		IF arrCheckListForNestedSymbols[uiCounterCheckSubItemsInContentOfDoc] = arrContentOfDocument[uiCounterCkeckContenInSubItems_1].sSymbolName THEN
			IF arrContentOfDocument[uiCounterCkeckContenInSubItems_1].arrSubItemSymbolType[uiCounterCkeckContenInSubItems_2] <> 'BOOL' AND arrContentOfDocument[uiCounterCkeckContenInSubItems_1].arrSubItemSymbolType[uiCounterCkeckContenInSubItems_2] <> 'BYTE' AND
				arrContentOfDocument[uiCounterCkeckContenInSubItems_1].arrSubItemSymbolType[uiCounterCkeckContenInSubItems_2] <> 'WORD' AND arrContentOfDocument[uiCounterCkeckContenInSubItems_1].arrSubItemSymbolType[uiCounterCkeckContenInSubItems_2] <> 'DWORD' AND
					arrContentOfDocument[uiCounterCkeckContenInSubItems_1].arrSubItemSymbolType[uiCounterCkeckContenInSubItems_2] <> 'SINT' AND arrContentOfDocument[uiCounterCkeckContenInSubItems_1].arrSubItemSymbolType[uiCounterCkeckContenInSubItems_2] <> 'USINT' AND
						arrContentOfDocument[uiCounterCkeckContenInSubItems_1].arrSubItemSymbolType[uiCounterCkeckContenInSubItems_2] <> 'INT' AND arrContentOfDocument[uiCounterCkeckContenInSubItems_1].arrSubItemSymbolType[uiCounterCkeckContenInSubItems_2] <> 'UINT' AND
							arrContentOfDocument[uiCounterCkeckContenInSubItems_1].arrSubItemSymbolType[uiCounterCkeckContenInSubItems_2] <> 'DINT' AND arrContentOfDocument[uiCounterCkeckContenInSubItems_1].arrSubItemSymbolType[uiCounterCkeckContenInSubItems_2] <> 'UDINT' AND
								arrContentOfDocument[uiCounterCkeckContenInSubItems_1].arrSubItemSymbolType[uiCounterCkeckContenInSubItems_2] <> 'LINT' AND arrContentOfDocument[uiCounterCkeckContenInSubItems_1].arrSubItemSymbolType[uiCounterCkeckContenInSubItems_2] <> 'ULINT' AND
									arrContentOfDocument[uiCounterCkeckContenInSubItems_1].arrSubItemSymbolType[uiCounterCkeckContenInSubItems_2] <> 'LWORD' AND arrContentOfDocument[uiCounterCkeckContenInSubItems_1].arrSubItemSymbolType[uiCounterCkeckContenInSubItems_2] <> 'REAL' AND
										arrContentOfDocument[uiCounterCkeckContenInSubItems_1].arrSubItemSymbolType[uiCounterCkeckContenInSubItems_2] <> 'LREAL' AND arrContentOfDocument[uiCounterCkeckContenInSubItems_1].arrSubItemSymbolType[uiCounterCkeckContenInSubItems_2] <> 'STRING(30)' AND
											arrContentOfDocument[uiCounterCkeckContenInSubItems_1].arrSubItemSymbolType[uiCounterCkeckContenInSubItems_2] <> 'TIME' AND arrContentOfDocument[uiCounterCkeckContenInSubItems_1].arrSubItemSymbolType[uiCounterCkeckContenInSubItems_2] <> 'TIME_OF_DAY' AND
												arrContentOfDocument[uiCounterCkeckContenInSubItems_1].arrSubItemSymbolType[uiCounterCkeckContenInSubItems_2] <> 'DATE' AND arrContentOfDocument[uiCounterCkeckContenInSubItems_1].arrSubItemSymbolType[uiCounterCkeckContenInSubItems_2] <> 'DATE_AND_TIME' AND 
			FIND(arrContentOfDocument[uiCounterCkeckContenInSubItems_1].arrSubItemSymbolType[uiCounterCkeckContenInSubItems_2],'OF BOOL') = 0 AND FIND(arrContentOfDocument[uiCounterCkeckContenInSubItems_1].arrSubItemSymbolType[uiCounterCkeckContenInSubItems_2],'OF BYTE') = 0 AND
				FIND(arrContentOfDocument[uiCounterCkeckContenInSubItems_1].arrSubItemSymbolType[uiCounterCkeckContenInSubItems_2],'OF WORD') = 0 AND FIND(arrContentOfDocument[uiCounterCkeckContenInSubItems_1].arrSubItemSymbolType[uiCounterCkeckContenInSubItems_2],'OF DWORD') = 0 AND
					FIND(arrContentOfDocument[uiCounterCkeckContenInSubItems_1].arrSubItemSymbolType[uiCounterCkeckContenInSubItems_2],'OF SINT') = 0 AND FIND(arrContentOfDocument[uiCounterCkeckContenInSubItems_1].arrSubItemSymbolType[uiCounterCkeckContenInSubItems_2],'OF USINT') = 0 AND 
						FIND(arrContentOfDocument[uiCounterCkeckContenInSubItems_1].arrSubItemSymbolType[uiCounterCkeckContenInSubItems_2],'OF INT') = 0 AND FIND(arrContentOfDocument[uiCounterCkeckContenInSubItems_1].arrSubItemSymbolType[uiCounterCkeckContenInSubItems_2],'OF UINT') = 0 AND
							FIND(arrContentOfDocument[uiCounterCkeckContenInSubItems_1].arrSubItemSymbolType[uiCounterCkeckContenInSubItems_2],'OF DINT') = 0 AND FIND(arrContentOfDocument[uiCounterCkeckContenInSubItems_1].arrSubItemSymbolType[uiCounterCkeckContenInSubItems_2],'OF UDINT') = 0 AND
								FIND(arrContentOfDocument[uiCounterCkeckContenInSubItems_1].arrSubItemSymbolType[uiCounterCkeckContenInSubItems_2],'OF LINT') = 0 AND FIND(arrContentOfDocument[uiCounterCkeckContenInSubItems_1].arrSubItemSymbolType[uiCounterCkeckContenInSubItems_2],'OF ULINT') = 0 AND
									FIND(arrContentOfDocument[uiCounterCkeckContenInSubItems_1].arrSubItemSymbolType[uiCounterCkeckContenInSubItems_2],'OF LWORD') = 0 AND FIND(arrContentOfDocument[uiCounterCkeckContenInSubItems_1].arrSubItemSymbolType[uiCounterCkeckContenInSubItems_2],'OF REAL') = 0 AND
										FIND(arrContentOfDocument[uiCounterCkeckContenInSubItems_1].arrSubItemSymbolType[uiCounterCkeckContenInSubItems_2],'OF LREAL') = 0 AND FIND(arrContentOfDocument[uiCounterCkeckContenInSubItems_1].arrSubItemSymbolType[uiCounterCkeckContenInSubItems_2],'OF STRING(30)') = 0 AND
											FIND(arrContentOfDocument[uiCounterCkeckContenInSubItems_1].arrSubItemSymbolType[uiCounterCkeckContenInSubItems_2],'OF TIME') = 0 AND FIND(arrContentOfDocument[uiCounterCkeckContenInSubItems_1].arrSubItemSymbolType[uiCounterCkeckContenInSubItems_2],'OF TIME_OF_DAY') = 0 AND
												FIND(arrContentOfDocument[uiCounterCkeckContenInSubItems_1].arrSubItemSymbolType[uiCounterCkeckContenInSubItems_2],'OF DATE') = 0 AND FIND(arrContentOfDocument[uiCounterCkeckContenInSubItems_1].arrSubItemSymbolType[uiCounterCkeckContenInSubItems_2],'OF DATE_AND_TIME') = 0 AND
			arrContentOfDocument[uiCounterCkeckContenInSubItems_1].arrSubItemSymbolType[uiCounterCkeckContenInSubItems_2] <> '' THEN 
				iStateParseDocument := 200;
					udiErrorCode := 117;
			END_IF	
		END_IF
		
		IF uiCounterCheckSubItemsInContentOfDoc >= uiCounterListForFBorStruct AND uiCounterCkeckContenInSubItems_1 >= uiCounterInProgressFromDocument AND uiCounterCkeckContenInSubItems_2 >= Constants_Communicator.uiArraySizeOfMarkedSubItems AND iStateParseDocument = 105 THEN 
			iStateParseDocument := 106; byProgress := byProgress + 1;
				uiCounterCheckSubItemsInContentOfDoc := 0; uiCounterCkeckContenInSubItems_1 := 0; uiCounterCkeckContenInSubItems_2 := 0;
		END_IF
		
	106://Check in Sub Items for no standart Datatypes in Array	
		uiCounterCkeckContenInSubItems_2 := uiCounterCkeckContenInSubItems_2 + 1;
		
		IF uiCounterCkeckContenInSubItems_2 > Constants_Communicator.uiArraySizeOfMarkedSubItems THEN uiCounterCkeckContenInSubItems_1 := uiCounterCkeckContenInSubItems_1 + 1; END_IF
			
		IF uiCounterCkeckContenInSubItems_2 > Constants_Communicator.uiArraySizeOfMarkedSubItems AND uiCounterCkeckContenInSubItems_1 > uiCounterInProgressFromDocument THEN uiCounterCheckSubItemsInContentOfDoc := uiCounterCheckSubItemsInContentOfDoc + 1; END_IF	

		IF uiCounterCkeckContenInSubItems_1 > uiCounterInProgressFromDocument THEN uiCounterCkeckContenInSubItems_1 := 1; END_IF	
		IF uiCounterCkeckContenInSubItems_2 > Constants_Communicator.uiArraySizeOfMarkedSubItems THEN uiCounterCkeckContenInSubItems_2 := 1; END_IF
	
		uiCounterCkeckContenInSubItems_2 := LIMIT(1,uiCounterCkeckContenInSubItems_2,Constants_Communicator.uiArraySizeOfMarkedSubItems);	
		uiCounterCheckSubItemsInContentOfDoc := LIMIT(1,uiCounterCheckSubItemsInContentOfDoc,Constants_Communicator.uiArraySizeOfSubItems);
		uiCounterCkeckContenInSubItems_1 := LIMIT(1,uiCounterCkeckContenInSubItems_1,Constants_Communicator.uiArraySizeOfSubItems);
		
		//Array with no Standart Datatype
		IF FIND(arrContentOfDocument[uiCounterCkeckContenInSubItems_1].arrSubItemSymbolType[uiCounterCkeckContenInSubItems_2],'ARRAY') = 1 AND 
			FIND(arrContentOfDocument[uiCounterCkeckContenInSubItems_1].arrSubItemSymbolType[uiCounterCkeckContenInSubItems_2],'OF BOOL') = 0 AND FIND(arrContentOfDocument[uiCounterCkeckContenInSubItems_1].arrSubItemSymbolType[uiCounterCkeckContenInSubItems_2],'OF BYTE') = 0 AND
				FIND(arrContentOfDocument[uiCounterCkeckContenInSubItems_1].arrSubItemSymbolType[uiCounterCkeckContenInSubItems_2],'OF WORD') = 0 AND FIND(arrContentOfDocument[uiCounterCkeckContenInSubItems_1].arrSubItemSymbolType[uiCounterCkeckContenInSubItems_2],'OF DWORD') = 0 AND
					FIND(arrContentOfDocument[uiCounterCkeckContenInSubItems_1].arrSubItemSymbolType[uiCounterCkeckContenInSubItems_2],'OF SINT') = 0 AND FIND(arrContentOfDocument[uiCounterCkeckContenInSubItems_1].arrSubItemSymbolType[uiCounterCkeckContenInSubItems_2],'OF USINT') = 0 AND 
						FIND(arrContentOfDocument[uiCounterCkeckContenInSubItems_1].arrSubItemSymbolType[uiCounterCkeckContenInSubItems_2],'OF INT') = 0 AND FIND(arrContentOfDocument[uiCounterCkeckContenInSubItems_1].arrSubItemSymbolType[uiCounterCkeckContenInSubItems_2],'OF UINT') = 0 AND
							FIND(arrContentOfDocument[uiCounterCkeckContenInSubItems_1].arrSubItemSymbolType[uiCounterCkeckContenInSubItems_2],'OF DINT') = 0 AND FIND(arrContentOfDocument[uiCounterCkeckContenInSubItems_1].arrSubItemSymbolType[uiCounterCkeckContenInSubItems_2],'OF UDINT') = 0 AND
								FIND(arrContentOfDocument[uiCounterCkeckContenInSubItems_1].arrSubItemSymbolType[uiCounterCkeckContenInSubItems_2],'OF LINT') = 0 AND FIND(arrContentOfDocument[uiCounterCkeckContenInSubItems_1].arrSubItemSymbolType[uiCounterCkeckContenInSubItems_2],'OF ULINT') = 0 AND
									FIND(arrContentOfDocument[uiCounterCkeckContenInSubItems_1].arrSubItemSymbolType[uiCounterCkeckContenInSubItems_2],'OF LWORD') = 0 AND FIND(arrContentOfDocument[uiCounterCkeckContenInSubItems_1].arrSubItemSymbolType[uiCounterCkeckContenInSubItems_2],'OF REAL') = 0 AND
										FIND(arrContentOfDocument[uiCounterCkeckContenInSubItems_1].arrSubItemSymbolType[uiCounterCkeckContenInSubItems_2],'OF LREAL') = 0 AND FIND(arrContentOfDocument[uiCounterCkeckContenInSubItems_1].arrSubItemSymbolType[uiCounterCkeckContenInSubItems_2],'OF STRING(30)') = 0 AND
											FIND(arrContentOfDocument[uiCounterCkeckContenInSubItems_1].arrSubItemSymbolType[uiCounterCkeckContenInSubItems_2],'OF TIME') = 0 AND FIND(arrContentOfDocument[uiCounterCkeckContenInSubItems_1].arrSubItemSymbolType[uiCounterCkeckContenInSubItems_2],'OF TIME_OF_DAY') = 0 AND
												FIND(arrContentOfDocument[uiCounterCkeckContenInSubItems_1].arrSubItemSymbolType[uiCounterCkeckContenInSubItems_2],'OF DATE') = 0 AND FIND(arrContentOfDocument[uiCounterCkeckContenInSubItems_1].arrSubItemSymbolType[uiCounterCkeckContenInSubItems_2],'OF DATE_AND_TIME') = 0 AND
			arrContentOfDocument[uiCounterCkeckContenInSubItems_1].arrSubItemSymbolType[uiCounterCkeckContenInSubItems_2] <> '' THEN 
				iStateParseDocument := 200;
					udiErrorCode := 118;
		END_IF
	
		IF uiCounterCheckSubItemsInContentOfDoc >= uiCounterListForFBorStruct AND uiCounterCkeckContenInSubItems_1 >= uiCounterInProgressFromDocument AND uiCounterCkeckContenInSubItems_2 >= Constants_Communicator.uiArraySizeOfMarkedSubItems AND iStateParseDocument = 106 THEN 
			iStateParseDocument := 0; byProgress := 100; bDone := TRUE; uiFoundItems := uiCounterInProgressFromDocument; 
		END_IF
		
	200://Error
		IF udiErrorCode = 101 OR udiErrorCode = 102 OR udiErrorCode = 103 OR udiErrorCode = 108 OR udiErrorCode = 109 OR udiErrorCode = 110 OR udiErrorCode = 3 OR udiErrorCode = 4 THEN sSymbolNameWithError := sSymbolName; END_IF
			IF udiErrorCode = 104 THEN sSymbolNameWithError := CONCAT(CONCAT(sSymbolName,'.'),sNameSubItem); END_IF 
				IF ((udiErrorCode = 111 OR udiErrorCode = 112) AND uiCounterWantedSymbolInProgress <= 1 AND uiSubItemArrayInProgress <= 2) THEN 
					sSymbolNameWithError := CONCAT(CONCAT(arrContentOfDocument[1].sSymbolName,'.'),arrContentOfDocument[1].arrSubItemName[1]); 
				END_IF
					IF ((udiErrorCode = 111 OR udiErrorCode = 112) AND uiCounterWantedSymbolInProgress > 1 AND uiSubItemArrayInProgress <= 2) THEN 
						sSymbolNameWithError := CONCAT(CONCAT(arrContentOfDocument[uiCounterWantedSymbolInProgress].sSymbolName,'.'),arrContentOfDocument[uiCounterWantedSymbolInProgress].arrSubItemName[1]); 
					END_IF
						IF ((udiErrorCode = 111 OR udiErrorCode = 112) AND uiCounterWantedSymbolInProgress <= 1 AND uiSubItemArrayInProgress > 2) THEN 
							sSymbolNameWithError := CONCAT(CONCAT(arrContentOfDocument[1].sSymbolName,'.'),arrContentOfDocument[1].arrSubItemName[uiSubItemArrayInProgress - 1]); 
						END_IF
							IF ((udiErrorCode = 111 OR udiErrorCode = 112) AND uiCounterWantedSymbolInProgress > 1 AND uiSubItemArrayInProgress > 2) THEN 
								sSymbolNameWithError := CONCAT(CONCAT(arrContentOfDocument[uiCounterWantedSymbolInProgress].sSymbolName,'.'),arrContentOfDocument[uiCounterWantedSymbolInProgress].arrSubItemName[uiSubItemArrayInProgress - 1]); 
							END_IF
								IF udiErrorCode = 115 OR udiErrorCode = 116 OR udiErrorCode = 117 THEN sSymbolNameWithError := arrCheckListForNestedSymbols[uiCounterCheckSubItemsInContentOfDoc]; END_IF 
									IF udiErrorCode = 118 THEN sSymbolNameWithError := arrContentOfDocument[uiCounterCkeckContenInSubItems_1].sSymbolName; END_IF 
		bError := TRUE;
			iStateParseDocument := 0;
			
END_CASE

//Save position
IF eSavePositionTMCFile = eSavePositionFile.ePostionC THEN fbFileOpen.sPathName := CONCAT(CONCAT('C:\TwinCAT\3.1\Config\TMC\',TwinCAT_SystemInfoVarList._AppInfo.ProjectName),'.tmc'); END_IF
IF eSavePositionTMCFile = eSavePositionFile.ePostionHardDisk THEN fbFileOpen.sPathName := CONCAT(CONCAT('Hard Disk\TwinCAT\3.1\Config\TMC\',TwinCAT_SystemInfoVarList._AppInfo.ProjectName),'.tmc'); END_IF

fbFileOpen(
	sNetId:= , 
	sPathName:= , 
	nMode:= FOPEN_MODEREAD OR FOPEN_MODETEXT, 
	ePath:= PATH_GENERIC, 
	bExecute:= , 
	tTimeout:= T#5S, 
	bBusy=> , 
	bError=> , 
	nErrId=> , 
	hFile=> );

FPErrorOpen(CLK:= fbFileOpen.bError, Q=> );
	
fbFileGet(
	sNetId:= , 
	hFile:= fbFileOpen.hFile, 
	bExecute:= , 
	tTimeout:= T#5S, 
	bBusy=> , 
	bError=> , 
	nErrId=> , 
	sLine=> , 
	bEOF=> );

FPErrorGet(CLK:= fbFileGet.bError, Q=> );

fbFileTell(
	sNetId:= , 
	hFile:= fbFileOpen.hFile, 
	bExecute:= , 
	tTimeout:= T#5S, 
	bBusy=> , 
	bError=> , 
	nErrId=> , 
	nSeekPos=> );

FPErrorTell(CLK:= fbFileTell.bError, Q=> );	

fbFileSeek(
	sNetId:= , 
	hFile:= fbFileOpen.hFile, 
	nSeekPos:= , 
	eOrigin:= SEEK_END, 
	bExecute:= , 
	tTimeout:= T#5S, 
	bBusy=> , 
	bError=> , 
	nErrId=> );

FPErrorSeek(CLK:= fbFileSeek.bError, Q=> );
	
fbFileClose(
	sNetId:= , 
	hFile:= fbFileOpen.hFile, 
	bExecute:= , 
	tTimeout:= T#5S, 
	bBusy=> , 
	bError=> , 
	nErrId=> );
	
FPErrorClose(CLK:= fbFileClose.bError, Q=> );	

//Progress
IF iStateParseDocument > 3 AND iStateParseDocument < 100 AND diEndPositionInDocument > 0 THEN
	byProgress := REAL_TO_BYTE(F_Scalvalue(x:= DINT_TO_REAL(fbFileTell.nSeekPos), x1:= 0, y1:= 0, x2:= DINT_TO_REAL(diEndPositionInDocument), y2:= 100));
		IF byProgress >= 5 THEN
			byProgress := byProgress - 5;
		ELSE
			byProgress := 0;
		END_IF
END_IF

END_FUNCTION_BLOCK

// ---- General/FUNs Internal/F_Scalvalue.TcPOU
{attribute 'conditionalshow'}
FUNCTION F_Scalvalue : REAL
VAR_INPUT
	{attribute 'hide'}
	x 	: REAL;		//Scale Value
	{attribute 'hide'}
	x1	: REAL;		//Point 1, x-coordinate
	{attribute 'hide'}
	y1	: REAL;		//Point 1, y-coordinate
	{attribute 'hide'}
	x2	: REAL;		//Point 2, x-coordinate
	{attribute 'hide'}
	y2	: REAL;		//Point 2, y-coordinate
END_VAR
VAR
	{attribute 'hide'}
	k, d: REAL;		//Calculation points
END_VAR

//Slope of the straight line
IF x2 <> x1 THEN
	k:=	(y2 - y1) / (x2 - x1);
ELSE
	//Avoid division by 0
	k:= 1;
END_IF
//Intersection with the Y axis
d:= y1 - (k * x1);

//Output scaling
F_Scalvalue:= (k * x) + d;

END_FUNCTION

// ---- Communicator/FBs Internal/FB_VarInfo_ErrorCodes.TcPOU
{attribute 'conditionalshow'}
FUNCTION_BLOCK FB_VarInfo_ErrorCodes
VAR_INPUT
	{attribute 'hide'}
	bErrorADS				: BOOL;											//Error ADS function
	{attribute 'hide'}
	bErrorIntern			: BOOL;											//Other Error
	{attribute 'hide'}
	udiErrorCodeADS			: UDINT;										//Error Code ADS function
	{attribute 'hide'}
	udiErrorCodesIntern		: UDINT;										//Error code from other errors
END_VAR
VAR_OUTPUT
	{attribute 'hide'}
	udiErrorCodeADS_Out		: UDINT;										//ADS return code
	{attribute 'hide'}
	bError					: BOOL;											//Error flag
	eErrorVarInfo_Out		: eErrorVarInfo;								//Enum with Error from the Var Info function
END_VAR
VAR
END_VAR

//Creator : Kai Ebensperger
//Company : Lynus AG
//Date : 01.04.2020
//Version : 1.0.0.0

//With this function its possible to give out a Error return code from the ads or the internal codes from the read variable info function
//Directly from the ads
IF bErrorIntern OR bErrorADS THEN bError := TRUE; ELSE bError := FALSE; END_IF
	IF bErrorADS THEN udiErrorCodeADS_Out := udiErrorCodeADS; ELSE udiErrorCodeADS_Out := 0; END_IF

//Internal error codes from Var Info
IF bErrorIntern AND udiErrorCodesIntern = 1 THEN eErrorVarInfo_Out := eErrorVarInfo.eArraySizeError; 
ELSIF bErrorIntern AND udiErrorCodesIntern = 2 THEN eErrorVarInfo_Out := eErrorVarInfo.eTimoutError;
ELSIF bErrorIntern AND udiErrorCodesIntern = 3 THEN eErrorVarInfo_Out := eErrorVarInfo.eCommentLenghtError;
ELSIF bErrorIntern AND udiErrorCodesIntern = 4 THEN eErrorVarInfo_Out := eErrorVarInfo.eCommentDescriptionError;
ELSIF bErrorIntern AND udiErrorCodesIntern = 5 THEN eErrorVarInfo_Out := eErrorVarInfo.eSymbolTypeError;
ELSIF bErrorIntern AND udiErrorCodesIntern = 6 THEN eErrorVarInfo_Out := eErrorVarInfo.eSymbolNameToLongError; 
ELSIF bErrorIntern AND udiErrorCodesIntern = 7 THEN eErrorVarInfo_Out := eErrorVarInfo.eReadWriteFunctionToMuch; 
ELSIF bErrorIntern AND udiErrorCodesIntern = 8 THEN eErrorVarInfo_Out := eErrorVarInfo.eVarInfoFunctionToMuch;
ELSIF bErrorIntern AND udiErrorCodesIntern = 9 THEN eErrorVarInfo_Out := eErrorVarInfo.eSendReceiveFunctionToMuch; 
ELSIF bErrorIntern AND udiErrorCodesIntern = 10 THEN eErrorVarInfo_Out := eErrorVarInfo.eMoreReadWriteFuctionsAsSymbols;
ELSIF bErrorIntern AND udiErrorCodesIntern = 11 THEN eErrorVarInfo_Out := eErrorVarInfo.eNoTMCFileSelected;
ELSIF bErrorIntern AND udiErrorCodesIntern = 12 THEN eErrorVarInfo_Out := eErrorVarInfo.eArrayWithNoStandartDatatype; 
ELSIF bErrorIntern AND udiErrorCodesIntern = 13 THEN eErrorVarInfo_Out := eErrorVarInfo.eSymbolNotFoundInTMCFile; 
ELSIF bErrorIntern AND udiErrorCodesIntern = 14 THEN eErrorVarInfo_Out := eErrorVarInfo.eSymbolNameWithSubItemIsToLong;	
ELSIF bErrorIntern AND udiErrorCodesIntern = 15 THEN eErrorVarInfo_Out := eErrorVarInfo.eToMuchSubItemsInSymbol;
ELSIF bErrorIntern AND udiErrorCodesIntern = 16 THEN eErrorVarInfo_Out := eErrorVarInfo.eToMuchSymbols;
ELSIF bErrorIntern AND udiErrorCodesIntern = 17 THEN eErrorVarInfo_Out := eErrorVarInfo.eSubItemsInfoError;
ELSIF bErrorIntern AND udiErrorCodesIntern = 18 THEN eErrorVarInfo_Out := eErrorVarInfo.eNoSendReceiveFunction;
ELSIF bErrorIntern AND udiErrorCodesIntern = 19 THEN eErrorVarInfo_Out := eErrorVarInfo.eNoReadWriteFunction;
ELSIF bErrorIntern AND udiErrorCodesIntern = 20 THEN eErrorVarInfo_Out := eErrorVarInfo.eNoSymbolsFound;	
//Internal error codes from Parse Function	
ELSIF bErrorIntern AND udiErrorCodesIntern = 100 THEN eErrorVarInfo_Out := eErrorVarInfo.eTMCFileTimoutError;
ELSIF bErrorIntern AND udiErrorCodesIntern = 101 THEN eErrorVarInfo_Out := eErrorVarInfo.eTMCFileContentOfSymbolIsToBig;
ELSIF bErrorIntern AND udiErrorCodesIntern = 102 THEN eErrorVarInfo_Out := eErrorVarInfo.eTMCFileSymbolNameToLongError;	
ELSIF bErrorIntern AND udiErrorCodesIntern = 103 THEN eErrorVarInfo_Out := eErrorVarInfo.eTMCFileToMuchSubItemsInOneSymbol;
ELSIF bErrorIntern AND udiErrorCodesIntern = 104 THEN eErrorVarInfo_Out := eErrorVarInfo.eTMCFileSubItemNameToLongError;
ELSIF bErrorIntern AND udiErrorCodesIntern = 105 THEN eErrorVarInfo_Out := eErrorVarInfo.eTMCFileErrorWhenOpeningTheFile;
ELSIF bErrorIntern AND udiErrorCodesIntern = 106 THEN eErrorVarInfo_Out := eErrorVarInfo.eTMCFileErrorWhenReadingTheFile;
ELSIF bErrorIntern AND udiErrorCodesIntern = 107 THEN eErrorVarInfo_Out := eErrorVarInfo.eTMCFileErrorWhenClosingTheFile;
ELSIF bErrorIntern AND udiErrorCodesIntern = 108 THEN eErrorVarInfo_Out := eErrorVarInfo.eTMCFileToMuchNoStandartDatatypes;	
ELSIF bErrorIntern AND udiErrorCodesIntern = 109 THEN eErrorVarInfo_Out := eErrorVarInfo.eTMCFileEnumNameToLongError;
ELSIF bErrorIntern AND udiErrorCodesIntern = 110 THEN eErrorVarInfo_Out := eErrorVarInfo.eTMCFileEnumIndexToMuchSizes;
ELSIF bErrorIntern AND udiErrorCodesIntern = 111 THEN eErrorVarInfo_Out := eErrorVarInfo.eTMCFileArraySizeError;
ELSIF bErrorIntern AND udiErrorCodesIntern = 112 THEN eErrorVarInfo_Out := eErrorVarInfo.eTMCFileStringSizeError;
ELSIF bErrorIntern AND udiErrorCodesIntern = 113 THEN eErrorVarInfo_Out := eErrorVarInfo.eTMCFileCheckPositionError;
ELSIF bErrorIntern AND udiErrorCodesIntern = 114 THEN eErrorVarInfo_Out := eErrorVarInfo.eTMCFileSearchPositionError;
ELSIF bErrorIntern AND udiErrorCodesIntern = 115 THEN eErrorVarInfo_Out := eErrorVarInfo.eTMCFileMissingSubItems;
ELSIF bErrorIntern AND udiErrorCodesIntern = 116 THEN eErrorVarInfo_Out := eErrorVarInfo.eTMCFileFunctionblockAccessNotAllowed;
ELSIF bErrorIntern AND udiErrorCodesIntern = 117 THEN eErrorVarInfo_Out := eErrorVarInfo.eTMCFileToMuchSubItemsInOtherSubItems;
ELSIF bErrorIntern AND udiErrorCodesIntern = 118 THEN eErrorVarInfo_Out := eErrorVarInfo.eTMCFileArrayWithNoStandartDatatype;
ELSE
	eErrorVarInfo_Out := eErrorVarInfo.eNoError;	
END_IF

END_FUNCTION_BLOCK

// ---- Communicator/FBs Internal/FB_VarReadWrite_ErrorCodes.TcPOU
{attribute 'conditionalshow'}
FUNCTION_BLOCK FB_VarReadWrite_ErrorCodes
VAR_INPUT
	{attribute 'hide'}
	bErrorADS					: BOOL;											//Error ADS function
	{attribute 'hide'}
	bErrorIntern				: BOOL;											//Other Error
	{attribute 'hide'}
	udiErrorCodeADS				: UDINT;										//Error Code ADS function
	{attribute 'hide'}
	udiErrorCodesInternRead		: UDINT;										//Error code from read function
	{attribute 'hide'}
	udiErrorCodesInternWrite	: UDINT;										//Error code from write function
END_VAR
VAR_OUTPUT
	{attribute 'hide'}
	udiErrorCodeADS_Out			: UDINT;										//ADS return code
	{attribute 'hide'}
	bError						: BOOL;											//Error flag
	eErrorReadWrite_Out			: eErrorReadWrite;								//Enum with Error from the Var read/write function
END_VAR
VAR
END_VAR

//Creator : Kai Ebensperger
//Company : Lynus AG
//Date : 20.04.2020
//Version : 1.0.0.0

//With this function its possible to give out a Error return code from the ads or the internal codes from the read/write variable function
//Directly from the ads
IF bErrorIntern OR bErrorADS THEN bError := TRUE; ELSE bError := FALSE; END_IF
	IF bErrorADS THEN udiErrorCodeADS_Out := udiErrorCodeADS; ELSE udiErrorCodeADS_Out := 0; END_IF

//Internal error codes
IF bErrorIntern AND udiErrorCodesInternRead = 0 THEN eErrorReadWrite_Out := eErrorReadWrite.eErrorRead; END_IF
IF bErrorIntern AND udiErrorCodesInternRead = 1 THEN eErrorReadWrite_Out := eErrorReadWrite.eErrorSizeFloatValueRead; END_IF
IF bErrorIntern AND udiErrorCodesInternWrite = 0 THEN eErrorReadWrite_Out := eErrorReadWrite.eErrorWrite; END_IF
IF bErrorIntern AND udiErrorCodesInternWrite = 1 THEN eErrorReadWrite_Out := eErrorReadWrite.eErrorSizeValueWrite; END_IF 
	IF NOT bErrorIntern AND NOT bErrorADS THEN
		eErrorReadWrite_Out := eErrorReadWrite.eNoError; 
	END_IF

END_FUNCTION_BLOCK

// ---- Energy/FBs Internal/Battery Inverter/FB_BatteryInverter.TcPOU
{attribute 'hide_all_locals'}
{attribute 'conditionalshow'}
FUNCTION_BLOCK FB_BatteryInverter
VAR_INPUT
	{attribute 'hide'}
	bEnable								: BOOL;								//Enable/Disable Battery Inverter
	{attribute 'hide'}
	bInverterOnOff						: BOOL;								//Switch the Inverter On or Off
	{attribute 'hide'}
	bError								: BOOL;								//Battery Inverter has a Error
	{attribute 'hide'}
	bWarning							: BOOL;								//Battery Inverter has a Warning
	{attribute 'hide'}
	bReset								: BOOL;								//Reset after the inverter switch off regarding a Error. Need also to reset the warning
	{attribute 'hide'}
	bWorkOnIslandMode					: BOOL;								//True when the inverter work in island mode
	{attribute 'hide'}
	bWriteWithDelay						: BOOL;								//Write with Delay the Data to the output (Not al Output Data is writen with Delay)
	{attribute 'hide'}
	byPriority							: BYTE; 							//Priority of the device if controlled via the EMS block => 1 2 3 (If 0 then this device does not exist for the EMS block)
	{attribute 'hide'}
	byReserveSOCEPO						: BYTE;								//Reserve SOC in battery for emergency power operation
	{attribute 'hide'}
	byMaxDepthOfDischargeEPO			: BYTE; 							//If islanding is active, the maximum discharge depth of the batteries can be set here until the inverter switches off.
	{attribute 'hide'}
	iErrorCode							: INT;								//Error Code from external Battery inverter
	{attribute 'hide'}
	iWarningCode						: INT;								//Warning Code from external Battery inverter
	{attribute 'hide'}
	dwBatterSOC							: DWORD;							//The actual Battery state of Charge
	{attribute 'hide'}
	rTargetPower						: REAL;								//Target Power from the EMS Function
	{attribute 'hide'}
	lrActualBatteryPower				: LREAL;							//Actual Battery power in W
	{attribute 'hide'}
	rMaxChargePowerBattInverter			: REAL; 							//Max. charge power battery inverter with unit W
	{attribute 'hide'}
	rMaxDischargePowerBattInverter		: REAL;								//Max. discharge power battery inverter with unit W
	{attribute 'hide'}
	lrBattInverterPowerOnIslandMode		: LREAL;							//Power from the battery inverter when island mode is active with unit W
	{attribute 'hide'}
	lrBattInverterPowerOnNormalMode		: LREAL;							//Power from the battery inverter when normal mode is active with unit W
	{attribute 'hide'}
	tTimDelayOutput						: TIME := T#5S;						//Delay Time to write some Data to the Output	
END_VAR
VAR_OUTPUT
	{attribute 'hide'}
	stDataBattInvertOut					: ST_BatteryInverter_Output;		//Batter Inverter output data
	{attribute 'hide'}
	stDataBattInvertOutDelay			: ST_BatteryInverter_Output;		//Batter Inverter output data with delay
END_VAR
VAR
	FPReset								: R_TRIG;							//Internal rising edge
	FPResetTim							: R_TRIG;							//Internal rising edge
	FPEnable							: R_TRIG;							//Internal positive Edge
	FNEnable							: F_TRIG;							//Internal negative Edge
	timReset							: TOF;								//Timer for Reset
	timStandby							: TON;								//Timer to set the inverter in standby mode
	timDisableInEPO						: TON;								//Timer do disable the inverter when work on Island mode an battery soc is under min
	timDelayOutputs						: TON;								//Timer to send Data with Delay to the outputs
	bMaxDephOfDischargeReached			: BOOL;								//True when the max of discharge in emergency power mode is reached
END_VAR

//Creator : Kai Ebensperger
//Company : Lynus AG
//Date : 18.05.2021
//Version : 1.0.0.0

//With this function is possible to control the most popular things on a battery inverter
//NOTE : With this Function its only poaaible to override the commands on a battery inverter
//All limits and important things control the inverter by himself.
//In Grid mode the Battery Inverter charge the battery to 100% SOC and discharge to 0% or to the limit for emergency power mode
//On Island mode the battery inverter charge the battery to 100% SOC. Discharge its possible to the max discharge setting. If the soc from the battery is <= this value the inverter switch off after 5 minutes when no power goes inside the battery
//With Reset you can reset the warnings and errors on the inverter.
//Also when the battery inverter is enabled by the timer for max discharge limit in emergency mode you can restart the inverter with a reset.
//When the target power for the inverter = 0 then the inverter go to the standby mode an switch off.

//---------------------------------------------------------------------Check the limits of the inputs--------------------------------------------------------------------------------------
byReserveSOCEPO := LIMIT(0,byReserveSOCEPO,100);
	byMaxDepthOfDischargeEPO := LIMIT(0,byMaxDepthOfDischargeEPO,100);
		dwBatterSOC := LIMIT(0,dwBatterSOC,100);
			rTargetPower := LIMIT(-100,rTargetPower,100);
				lrActualBatteryPower := LIMIT(-1000000,lrActualBatteryPower,1000000);
					lrBattInverterPowerOnIslandMode := LIMIT(-1000000,lrBattInverterPowerOnIslandMode,1000000);
						lrBattInverterPowerOnNormalMode := LIMIT(-1000000,lrBattInverterPowerOnNormalMode,1000000);
							rMaxChargePowerBattInverter := LIMIT(-1000000,rMaxChargePowerBattInverter,1000000);
								rMaxDischargePowerBattInverter := LIMIT(-1000000,rMaxDischargePowerBattInverter,1000000);

//---------------------------------------------------------------------------Data directly to the output-------------------------------------------------------------------------------------------
stDataBattInvertOut.byPriority := byPriority;
	stDataBattInvertOut.bEnabled := bEnable;
		stDataBattInvertOut.bWorkOnIslandMode := bWorkOnIslandMode;

//--------------------------------------------------------------------------Max Deph of discharge SOC in Emergency power mode---------------------------------------------------------------
IF dwBatterSOC <= byMaxDepthOfDischargeEPO AND lrActualBatteryPower >= 0 AND stDataBattInvertOut.bWorkOnIslandMode THEN timDisableInEPO.IN := TRUE; END_IF
	IF dwBatterSOC > byMaxDepthOfDischargeEPO OR lrActualBatteryPower < 0 OR NOT stDataBattInvertOut.bWorkOnIslandMode OR NOT stDataBattInvertOut.bOnOff OR (FPResetTim.Q AND bMaxDephOfDischargeReached) THEN timDisableInEPO.IN := FALSE; bMaxDephOfDischargeReached := FALSE; END_IF	
		timDisableInEPO(IN:= , PT:= T#5M, Q=> , ET=> );  
			IF timDisableInEPO.Q THEN bMaxDephOfDischargeReached := TRUE; END_IF		
		
//-----------------------------------------------------------------------------Reset-------------------------------------------------------------------------------------------------------
FPReset(CLK:= bReset, Q=> );
	timReset(IN:= stDataBattInvertOut.byErrorWarning <> 0 AND FPReset.Q AND NOT timReset.Q, PT:= T#2S, Q=> stDataBattInvertOut.bStateReset, ET=> );
		FPResetTim(CLK:= timReset.Q, Q=> );
			IF FPResetTim.Q THEN stDataBattInvertOut.byErrorWarning := 0; END_IF	

//--------------------------------------------------------------------------Error or Warning-------------------------------------------------------------------------------------------------
IF bWarning AND stDataBattInvertOut.byErrorWarning <> 2 THEN stDataBattInvertOut.byErrorWarning := 1; END_IF 
IF bError OR (timDisableInEPO.Q AND NOT FPResetTim.Q) THEN stDataBattInvertOut.byErrorWarning := 2; END_IF 			

//Error Codes
IF stDataBattInvertOut.byErrorWarning = 2 AND iErrorCode = 0 THEN stDataBattInvertOut.eMessage := E_Message_BatteryInverter.eBatteryInverterError;
ELSIF stDataBattInvertOut.byErrorWarning = 2 AND iErrorCode = 1 THEN stDataBattInvertOut.eMessage := E_Message_BatteryInverter.eTooMuchBatteryInverter;
ELSE stDataBattInvertOut.eMessage := E_Message_BatteryInverter.eNoMessage; 
END_IF
			
//--------------------------------------------------------------------------Target power--------------------------------------------------------------------------------------------------
stDataBattInvertOut.rTargetPower := rTargetPower;
	//Target power to 0
	IF (NOT stDataBattInvertOut.bWorkOnIslandMode AND stDataBattInvertOut.rTargetPower > 0 AND dwBatterSOC <= byReserveSOCEPO) OR
		(stDataBattInvertOut.rTargetPower < 0 AND dwBatterSOC >= 100) OR
			(NOT stDataBattInvertOut.bWorkOnIslandMode AND stDataBattInvertOut.rTargetPower > 0 AND dwBatterSOC <= 0) THEN 
				stDataBattInvertOut.rTargetPower := 0; 
	END_IF  
		//Set the Inverter in Standby	
		timStandby(IN:= stDataBattInvertOut.rTargetPower = 0 AND NOT stDataBattInvertOut.bWorkOnIslandMode, PT:= T#1M, Q=> , ET=> );
	
//--------------------------------------------------------------------Enable or disable the Inverter--------------------------------------------------------------------------------------
IF bEnable AND bInverterOnOff AND stDataBattInvertOut.byErrorWarning <> 2 THEN
	stDataBattInvertOut.bOnOff := TRUE;
END_IF			
	IF timStandby.Q OR stDataBattInvertOut.byErrorWarning = 2 OR NOT bEnable OR NOT bInverterOnOff THEN
		stDataBattInvertOut.bOnOff := FALSE;
	END_IF 				
	
//-------------------------------------------------------------------Outputs--------------------------------------------------------------------------------------------------------------
IF stDataBattInvertOut.bWorkOnIslandMode THEN 
	stDataBattInvertOut.lrPowerOnIslandMode := lrBattInverterPowerOnIslandMode / 1000;
		stDataBattInvertOut.lrPowerOnIslandMode := LINT_TO_LREAL(LREAL_TO_LINT(stDataBattInvertOut.lrPowerOnIslandMode * 100)) / 100;
			stDataBattInvertOut.lrPowerNormalMode := 0;	 
ELSE
	stDataBattInvertOut.lrPowerNormalMode := lrBattInverterPowerOnNormalMode / 1000;
		stDataBattInvertOut.lrPowerNormalMode := LINT_TO_LREAL(LREAL_TO_LINT(stDataBattInvertOut.lrPowerNormalMode * 100)) / 100; 	 
			stDataBattInvertOut.lrPowerOnIslandMode := 0;
END_IF

stDataBattInvertOut.rMaxChargePower := rMaxChargePowerBattInverter / 1000;
	stDataBattInvertOut.rMaxChargePower := DINT_TO_REAL(REAL_TO_DINT(stDataBattInvertOut.rMaxChargePower * 100)) / 100; 
	
stDataBattInvertOut.rMaxDischargePower := rMaxDischargePowerBattInverter / 1000;
	stDataBattInvertOut.rMaxDischargePower := DINT_TO_REAL(REAL_TO_DINT(stDataBattInvertOut.rMaxDischargePower * 100)) / 100; 

timDelayOutputs(IN:= bWriteWithDelay AND bEnable AND NOT timDelayOutputs.Q, PT:= tTimDelayOutput, Q=> , ET=> );
	FPEnable(CLK:= bEnable, Q=> );
		FNEnable(CLK:= bEnable, Q=> );
		
//Write with Delay or without
IF (bWriteWithDelay AND (timDelayOutputs.Q OR FPEnable.Q OR FNEnable.Q)) OR NOT bWriteWithDelay THEN
	stDataBattInvertOutDelay := stDataBattInvertOut;	
END_IF

END_FUNCTION_BLOCK

// ---- Energy/FBs Internal/Battery Inverter/FB_BatteryInverter_11.TcPOU
{attribute 'hide_all_locals'}
{attribute 'conditionalshow'}
FUNCTION_BLOCK FB_BatteryInverter_11
VAR_INPUT
	{attribute 'hide'}
	bEnable								: BOOL;								//Enable/Disable Battery Inverter
	{attribute 'hide'}
	bInverterOnOff						: BOOL;								//Switch the Inverter On or Off
	{attribute 'hide'}
	bError								: BOOL;								//Battery Inverter has a Error
	{attribute 'hide'}
	bWarning							: BOOL;								//Battery Inverter has a Warning
	{attribute 'hide'}
	bReset								: BOOL;								//Reset after the inverter switch off regarding a Error. Need also to reset the warning
	{attribute 'hide'}
	bWorkOnIslandMode					: BOOL;								//True when the inverter work in island mode
	{attribute 'hide'}
	bWriteWithDelay						: BOOL;								//Write with Delay the Data to the output (Not al Output Data is writen with Delay)
	{attribute 'hide'}
	byPriority							: BYTE; 							//Priority of the device if controlled via the EMS block => 1 2 3 (If 0 then this device does not exist for the EMS block)
	{attribute 'hide'}
	byReserveSOCEPO						: BYTE;								//Reserve SOC in battery for emergency power operation
	{attribute 'hide'}
	byMaxDepthOfDischargeEPO			: BYTE; 							//If islanding is active, the maximum discharge depth of the batteries can be set here until the inverter switches off.
	{attribute 'hide'}
	iErrorCode							: INT;								//Error Code from external Battery inverter
	{attribute 'hide'}
	iWarningCode						: INT;								//Warning Code from external Battery inverter
	{attribute 'hide'}
	dwBatterSOC							: DWORD;							//The actual Battery state of Charge
	{attribute 'hide'}
	rTargetPower						: REAL;								//Target Power from the EMS Function
	{attribute 'hide'}
	lrActualBatteryPower				: LREAL;							//Actual Battery power in W
	{attribute 'hide'}
	rMaxChargePowerBattInverter			: REAL; 							//Max. charge power battery inverter with unit W
	{attribute 'hide'}
	rMaxDischargePowerBattInverter		: REAL;								//Max. discharge power battery inverter with unit W
	{attribute 'hide'}
	lrBattInverterPowerOnIslandMode		: LREAL;							//Power from the battery inverter when island mode is active with unit W
	{attribute 'hide'}
	lrBattInverterPowerOnNormalMode		: LREAL;							//Power from the battery inverter when normal mode is active with unit W
	{attribute 'hide'}
	tTimDelayOutput						: TIME := T#5S;						//Delay Time to write some Data to the Output	
	by_minDischargeSOC					: BYTE;								//minimum SOC to discharge too
	by_maxChargeSOC						: BYTE;								//maximum SOC to charge too
END_VAR
VAR_OUTPUT
	{attribute 'hide'}
	stDataBattInvertOut					: ST_BatteryInverter_Output;		//Batter Inverter output data
	{attribute 'hide'}
	stDataBattInvertOutDelay			: ST_BatteryInverter_Output;		//Batter Inverter output data with delay
END_VAR
VAR
	FPReset								: R_TRIG;							//Internal rising edge
	FPResetTim							: R_TRIG;							//Internal rising edge
	FPEnable							: R_TRIG;							//Internal positive Edge
	FNEnable							: F_TRIG;							//Internal negative Edge
	timReset							: TOF;								//Timer for Reset
	timStandby							: TON;								//Timer to set the inverter in standby mode
	timDisableInEPO						: TON;								//Timer do disable the inverter when work on Island mode an battery soc is under min
	timDelayOutputs						: TON;								//Timer to send Data with Delay to the outputs
	bMaxDephOfDischargeReached			: BOOL;								//True when the max of discharge in emergency power mode is reached
END_VAR

//Creator : Stefan Lackner (based on Kai Ebensperger V1.0.0.0)
//Company : EfficientIO
//Date : 21.03.2024
//Version : 1.1.0.0

//With this function is possible to control the most popular things on a battery inverter
//NOTE : With this Function its only poaaible to override the commands on a battery inverter
//All limits and important things control the inverter by himself.
//In Grid mode the Battery Inverter charge the battery to 100% SOC and discharge to 0% or to the limit for emergency power mode
//On Island mode the battery inverter charge the battery to 100% SOC. Discharge its possible to the max discharge setting. If the soc from the battery is <= this value the inverter switch off after 5 minutes when no power goes inside the battery
//With Reset you can reset the warnings and errors on the inverter.
//Also when the battery inverter is enabled by the timer for max discharge limit in emergency mode you can restart the inverter with a reset.
//When the target power for the inverter = 0 then the inverter go to the standby mode an switch off.

// V1.1 added max/min SOC charge value
//---------------------------------------------------------------------Check the limits of the inputs--------------------------------------------------------------------------------------
byReserveSOCEPO := LIMIT(0,byReserveSOCEPO,100);
byMaxDepthOfDischargeEPO := LIMIT(0,byMaxDepthOfDischargeEPO,100);
dwBatterSOC := LIMIT(0,dwBatterSOC,100);
rTargetPower := LIMIT(-100,rTargetPower,100);
lrActualBatteryPower := LIMIT(-1000000,lrActualBatteryPower,1000000);
lrBattInverterPowerOnIslandMode := LIMIT(-1000000,lrBattInverterPowerOnIslandMode,1000000);
lrBattInverterPowerOnNormalMode := LIMIT(-1000000,lrBattInverterPowerOnNormalMode,1000000);
rMaxChargePowerBattInverter := LIMIT(-1000000,rMaxChargePowerBattInverter,1000000);
rMaxDischargePowerBattInverter := LIMIT(-1000000,rMaxDischargePowerBattInverter,1000000);
by_maxChargeSOC := LIMIT (1,by_maxChargeSOC,100);

//---------------------------------------------------------------------------Data directly to the output-------------------------------------------------------------------------------------------
stDataBattInvertOut.byPriority := byPriority;
stDataBattInvertOut.bEnabled := bEnable;
stDataBattInvertOut.bWorkOnIslandMode := bWorkOnIslandMode;

//--------------------------------------------------------------------------Max Deph of discharge SOC in Emergency power mode---------------------------------------------------------------
IF dwBatterSOC <= byMaxDepthOfDischargeEPO AND lrActualBatteryPower >= 0 AND stDataBattInvertOut.bWorkOnIslandMode THEN 
	timDisableInEPO.IN := TRUE; 
END_IF
IF dwBatterSOC > byMaxDepthOfDischargeEPO OR lrActualBatteryPower < 0 OR NOT stDataBattInvertOut.bWorkOnIslandMode OR NOT stDataBattInvertOut.bOnOff OR (FPResetTim.Q AND bMaxDephOfDischargeReached) THEN 
	timDisableInEPO.IN := FALSE; 
	bMaxDephOfDischargeReached := FALSE; 
END_IF	
timDisableInEPO(	IN:= , 
					PT:= T#5M, 
					Q=> , 
					ET=> );  
IF timDisableInEPO.Q THEN 
	bMaxDephOfDischargeReached := TRUE; 
END_IF		
		
//-----------------------------------------------------------------------------Reset-------------------------------------------------------------------------------------------------------
FPReset(	CLK:= bReset, 
			Q=> );
timReset(	IN:= stDataBattInvertOut.byErrorWarning <> 0 AND FPReset.Q AND NOT timReset.Q, 
			PT:= T#2S, 
			Q=> stDataBattInvertOut.bStateReset, 
			ET=> );
FPResetTim(	CLK:= timReset.Q, 
			Q=> );
IF FPResetTim.Q THEN 
	stDataBattInvertOut.byErrorWarning := 0; 
END_IF	

//--------------------------------------------------------------------------Error or Warning-------------------------------------------------------------------------------------------------
IF bWarning AND stDataBattInvertOut.byErrorWarning <> 2 THEN 
	stDataBattInvertOut.byErrorWarning := 1; 
END_IF 
IF bError OR (timDisableInEPO.Q AND NOT FPResetTim.Q) THEN 
	stDataBattInvertOut.byErrorWarning := 2; 
END_IF 			

//Error Codes
IF stDataBattInvertOut.byErrorWarning = 2 AND iErrorCode = 0 THEN 
	stDataBattInvertOut.eMessage := E_Message_BatteryInverter.eBatteryInverterError;
ELSIF stDataBattInvertOut.byErrorWarning = 2 AND iErrorCode = 1 THEN
	stDataBattInvertOut.eMessage := E_Message_BatteryInverter.eTooMuchBatteryInverter;
ELSE 
	stDataBattInvertOut.eMessage := E_Message_BatteryInverter.eNoMessage; 
END_IF
			
//--------------------------------------------------------------------------Target power--------------------------------------------------------------------------------------------------
stDataBattInvertOut.rTargetPower := rTargetPower;
//Target power to 0
IF (NOT stDataBattInvertOut.bWorkOnIslandMode AND stDataBattInvertOut.rTargetPower > 0 AND dwBatterSOC <= byReserveSOCEPO) OR
(stDataBattInvertOut.rTargetPower < 0 AND dwBatterSOC >= by_maxChargeSOC) OR
(NOT stDataBattInvertOut.bWorkOnIslandMode AND stDataBattInvertOut.rTargetPower > 0 AND dwBatterSOC <= 0) OR
(stDataBattInvertOut.rTargetPower > 0 AND dwBatterSOC <= by_minDischargeSOC) THEN 
	stDataBattInvertOut.rTargetPower := 0; 
END_IF  
//Set the Inverter in Standby	
timStandby(	IN:= stDataBattInvertOut.rTargetPower = 0 AND NOT stDataBattInvertOut.bWorkOnIslandMode, 
			PT:= T#1M, 
			Q=> , 
			ET=> );

//--------------------------------------------------------------------Enable or disable the Inverter--------------------------------------------------------------------------------------
IF bEnable AND bInverterOnOff AND stDataBattInvertOut.byErrorWarning <> 2 THEN
	stDataBattInvertOut.bOnOff := TRUE;
END_IF			
IF timStandby.Q OR stDataBattInvertOut.byErrorWarning = 2 OR NOT bEnable OR NOT bInverterOnOff THEN
	stDataBattInvertOut.bOnOff := FALSE;
END_IF 				
	
//-------------------------------------------------------------------Outputs--------------------------------------------------------------------------------------------------------------
IF stDataBattInvertOut.bWorkOnIslandMode THEN 
	stDataBattInvertOut.lrPowerOnIslandMode := lrBattInverterPowerOnIslandMode / 1000;
	stDataBattInvertOut.lrPowerOnIslandMode := LINT_TO_LREAL(LREAL_TO_LINT(stDataBattInvertOut.lrPowerOnIslandMode * 100)) / 100;
	stDataBattInvertOut.lrPowerNormalMode := 0;	 
ELSE
	stDataBattInvertOut.lrPowerNormalMode := lrBattInverterPowerOnNormalMode / 1000;
	stDataBattInvertOut.lrPowerNormalMode := LINT_TO_LREAL(LREAL_TO_LINT(stDataBattInvertOut.lrPowerNormalMode * 100)) / 100; 	 
	stDataBattInvertOut.lrPowerOnIslandMode := 0;
END_IF

stDataBattInvertOut.rMaxChargePower := rMaxChargePowerBattInverter / 1000;
stDataBattInvertOut.rMaxChargePower := DINT_TO_REAL(REAL_TO_DINT(stDataBattInvertOut.rMaxChargePower * 100)) / 100; 
	
stDataBattInvertOut.rMaxDischargePower := rMaxDischargePowerBattInverter / 1000;
stDataBattInvertOut.rMaxDischargePower := DINT_TO_REAL(REAL_TO_DINT(stDataBattInvertOut.rMaxDischargePower * 100)) / 100; 

timDelayOutputs(	IN:= bWriteWithDelay AND bEnable AND NOT timDelayOutputs.Q, 
					PT:= tTimDelayOutput, 
					Q=> , 
					ET=> );
FPEnable(	CLK:= bEnable, 
			Q=> );
FNEnable(	CLK:= bEnable, 
			Q=> );
		
//Write with Delay or without
IF (bWriteWithDelay AND (timDelayOutputs.Q OR FPEnable.Q OR FNEnable.Q)) OR NOT bWriteWithDelay THEN
	stDataBattInvertOutDelay := stDataBattInvertOut;	
END_IF

END_FUNCTION_BLOCK

// ---- Energy/FBs Internal/Battery/FB_Battery.TcPOU
{attribute 'hide_all_locals'}
{attribute 'conditionalshow'}
FUNCTION_BLOCK FB_Battery
VAR_INPUT
	{attribute 'hide'}
	bEnable								: BOOL;					//Enable this function
	{attribute 'hide'}
	bError								: BOOL;					//Battery has a error
	{attribute 'hide'}
	bWarning							: BOOL;					//Battery has a warning
	{attribute 'hide'}
	bCalculatePower						: BOOL;					//When its true, then calculate the power with then battery voltage and the battery current
	{attribute 'hide'}
	bReset								: BOOL;					//Reset the Error and the warning
	{attribute 'hide'}
	bWriteWithDelay						: BOOL;					//Write with Delay the Data to the output (Not al Output Data is writen with Delay)
	{attribute 'hide'}
	iErrorCode							: INT;					//Error Code from external Batterysystem
	{attribute 'hide'}
	iWarningCode						: INT;					//Warning Code from external Batterysystem
	{attribute 'hide'}
	dwBatterySOC						: DWORD;				//The actual Battery state of Charge
	{attribute 'hide'}
	dwBatterySOH						: DWORD;				//The actual battery state of health
	{attribute 'hide'}
	rBatteryVoltage						: REAL;					//Battery Voltage with Unit V
	{attribute 'hide'}
	rMaxDcChargeCurrentBattery			: REAL;					//Max. dc charge current battery with unit A 
	{attribute 'hide'}
	rMaxDcDischargeCurrentBattery		: REAL;					//Max. dc discharge current battery with unit A
	{attribute 'hide'}
	rMaxChargeVoltage					: REAL;					//Max. charge voltage from the battery with unit V
	{attribute 'hide'}
	lrMaxCapacityBattery				: LREAL;				//Max capacity from the Battery 
	{attribute 'hide'}
	lrBatteryPower						: LREAL;				//Battery Power with unit W
	{attribute 'hide'}
	lrBatteryCurrent					: LREAL;				//Battery current with unit A
	{attribute 'hide'}
	lrBatteryTemp						: LREAL;				//Battery temperarure with unit °C
	{attribute 'hide'}
	tTimDelayOutput						: TIME := T#5S;			//Delay Time to write some Data to the Output
END_VAR
VAR_OUTPUT
	{attribute 'hide'}
	stDataBatteryOut					: ST_Battery_Output;	//Output Data from the batter
	{attribute 'hide'}
	stDataBatteryOutDelay				: ST_Battery_Output;	//Output Data from the batter with delay
END_VAR
VAR
	FPReset								: R_TRIG;				//Internal positive edge
	FPEnable							: R_TRIG;				//Internal positive Edge
	FNEnable							: F_TRIG;				//Internal negative Edge
	timDelayOutputs						: TON;					//Timer to send Data with Delay to the outputs
END_VAR

//Creator : Kai Ebensperger
//Company : Lynus AG
//Date : 18.05.2021
//Version : 1.0.0.0

//With this function is possible to read in the most popular values from a battery
//The function calculate the actual capacity from the battery in kWh

//---------------------------------------------------------------------Check the limits of the inputs--------------------------------------------------------------------------------------

dwBatterySOC := LIMIT(0,dwBatterySOC,100);
	dwBatterySOH := LIMIT(0,dwBatterySOH,100);	
		rBatteryVoltage := LIMIT(0,rBatteryVoltage,1000);	
			rMaxDcChargeCurrentBattery := LIMIT(0,rMaxDcChargeCurrentBattery,10000);
				rMaxDcDischargeCurrentBattery := LIMIT(0,rMaxDcDischargeCurrentBattery,10000);
					rMaxChargeVoltage := LIMIT(0,rMaxChargeVoltage,1000);
						lrMaxCapacityBattery := LIMIT(0,lrMaxCapacityBattery,1000);
							lrBatteryPower := LIMIT(-1000000,lrBatteryPower,1000000);
								lrBatteryCurrent := LIMIT(-10000,lrBatteryCurrent,10000);
									lrBatteryTemp := LIMIT(-40,lrBatteryTemp,150);

//----------------------------------------------------------------------------Power from the battery-----------------------------------------------------------------------------------------------
IF bCalculatePower THEN 
	stDataBatteryOut.lrPower := (rBatteryVoltage * lrBatteryCurrent) / 1000; 
ELSE
	stDataBatteryOut.lrPower := lrBatteryPower / 1000;
END_IF

stDataBatteryOut.lrPower := LINT_TO_LREAL(LREAL_TO_LINT(stDataBatteryOut.lrPower * 100)) / 100;	

//Battery charge
IF stDataBatteryOut.lrPower < 0 THEN 
	stDataBatteryOut.lrPowerConsumption := stDataBatteryOut.lrPower * - 1;
	stDataBatteryOut.lrPowerProduction := 0;
END_IF
//Battery discharge
IF stDataBatteryOut.lrPower > 0 THEN 
	stDataBatteryOut.lrPowerConsumption := 0;
	stDataBatteryOut.lrPowerProduction := stDataBatteryOut.lrPower;
END_IF
//Power = 0
IF stDataBatteryOut.lrPower = 0 THEN 
	stDataBatteryOut.lrPowerConsumption := 0;
	stDataBatteryOut.lrPowerProduction := 0;
END_IF

//----------------------------------------------------------------------------Battery capacity-----------------------------------------------------------------------------------------------------

stDataBatteryOut.lrCapacity := (lrMaxCapacityBattery * dwBatterySOC) / 100; 
	stDataBatteryOut.lrCapacity := LINT_TO_LREAL(LREAL_TO_LINT(stDataBatteryOut.lrCapacity * 100)) / 100;	
								
//---------------------------------------------------------------------------Data directly to the output-------------------------------------------------------------------------------------------

stDataBatteryOut.bEnabled := bEnable;

IF bEnable THEN
	stDataBatteryOut.dwSOC := dwBatterySOC;
		stDataBatteryOut.dwSOH := dwBatterySOH;
			stDataBatteryOut.rBatteryVoltage := DINT_TO_REAL(REAL_TO_DINT(rBatteryVoltage * 100)) / 100; 
				stDataBatteryOut.rMaxDcChargeCurrent:= DINT_TO_REAL(REAL_TO_DINT(rMaxDcChargeCurrentBattery * 100)) / 100;
					stDataBatteryOut.rMaxDcDischargeCurrent := DINT_TO_REAL(REAL_TO_DINT(rMaxDcDischargeCurrentBattery * 100)) / 100;
						stDataBatteryOut.rMaxChargeVoltage := DINT_TO_REAL(REAL_TO_DINT(rMaxChargeVoltage * 100)) / 100;	
							stDataBatteryOut.lrCurrent := LINT_TO_LREAL(LREAL_TO_LINT(lrBatteryCurrent * 100)) / 100;
								stDataBatteryOut.lrTemp := LINT_TO_LREAL(LREAL_TO_LINT(lrBatteryTemp * 100)) / 100;	
ELSE
	stDataBatteryOut.dwSOC := 0;
		stDataBatteryOut.dwSOH := 0;
			stDataBatteryOut.rBatteryVoltage := 0; 
				stDataBatteryOut.rMaxDcChargeCurrent := 0;
					stDataBatteryOut.rMaxDcDischargeCurrent := 0;
						stDataBatteryOut.rMaxChargeVoltage := 0;	
							stDataBatteryOut.lrCurrent := 0;
								stDataBatteryOut.lrTemp := 0;
									stDataBatteryOut.lrCapacity := 0;
										stDataBatteryOut.lrPower := 0;
											stDataBatteryOut.lrPowerConsumption := 0;
												stDataBatteryOut.lrPowerProduction := 0;	
END_IF

//--------------------------------------------------------------------------Error or Warning-------------------------------------------------------------------------------------------------

FPReset(CLK:= bReset, Q=> );
	IF FPReset.Q THEN stDataBatteryOut.byErrorWarning := 0; END_IF

IF bWarning AND stDataBatteryOut.byErrorWarning <> 2 THEN stDataBatteryOut.byErrorWarning := 1; END_IF
IF bError THEN stDataBatteryOut.byErrorWarning := 2; END_IF

//Error Codes
IF stDataBatteryOut.byErrorWarning = 2 AND iErrorCode = 0 THEN stDataBatteryOut.eMessage := E_Message_Battery.eBatteryError;
ELSIF stDataBatteryOut.byErrorWarning = 2 AND iErrorCode = 1 THEN stDataBatteryOut.eMessage := E_Message_Battery.eTooMuchBattery;
ELSE stDataBatteryOut.eMessage := E_Message_Battery.eNoMessage; 
END_IF

//---------------------------------------------------------------Outputs-------------------------------------------------------------------------------*)

timDelayOutputs(IN:= bWriteWithDelay AND bEnable AND NOT timDelayOutputs.Q, PT:= tTimDelayOutput, Q=> , ET=> );
	FPEnable(CLK:= bEnable, Q=> );
		FNEnable(CLK:= bEnable, Q=> );
		
//Write with Delay or without
IF (bWriteWithDelay AND (timDelayOutputs.Q OR FPEnable.Q OR FNEnable.Q)) OR NOT bWriteWithDelay THEN
	stDataBatteryOutDelay := stDataBatteryOut;
END_IF

END_FUNCTION_BLOCK

// ---- Energy/FBs Internal/Beckhoff/FB_KL3403_SimpleProcessImage.TcPOU
{attribute 'conditionalshow'}
FUNCTION_BLOCK FB_KL3403_SimpleProcessImage
VAR_INPUT
	{attribute 'hide'}
	uiKBusState_IN						: UINT;							//K-Bus State from the K-Bus Box on wich the Terminal is connected. (Connect with FB_K_Bus_state)
	{attribute 'hide'}
	uiCurrentTransformerRatioL1			: UINT;							//Current Transformer Ratio for Channel 1 (L1)
	{attribute 'hide'}
	uiCurrentTransformerRatioL2			: UINT;							//Current Transformer Ratio for Channel 2 (L2)
	{attribute 'hide'}
	uiCurrentTransformerRatioL3			: UINT;							//Current Transformer Ratio for Channel 3 (L3)
	{attribute 'hide'}
	rResolutionCurrent					: REAL := 0.001;				//Resolution for the Current
	{attribute 'hide'}
	rResolutionPower					: REAL := 0.1;					//Resolution for the Power
	{attribute 'hide'}
	rResolutionEnergy					: REAL := 0.01;					//Resolution for the Energy	
END_VAR
VAR_OUTPUT
	{attribute 'hide'}
	stDataL1							: ST_KL3403;					//Data from Channel 1 (L1)
	{attribute 'hide'}
	stDataL2							: ST_KL3403;					//Data from Channel 2 (L2)
	{attribute 'hide'}
	stDataL3							: ST_KL3403;					//Data from Channel 3 (L3)
END_VAR
VAR
	{attribute 'hide'}
	timActive							: TON;							//Timer to activate the Statemachine
	{attribute 'hide'}
	timTimeout							: TON;							//Timeout Timer for the State Machine
	{attribute 'hide'}
	arrDataOk							: ARRAY[1..3] OF BOOL;			//Array with the Information if the Data In deliver all Information from each channel
	{attribute 'hide'}
	bErrorTimeOut						: BOOL;							//timout Error
	{attribute 'hide'}
	iState								: INT;							//Variable for the Statemachine
	{attribute 'hide'}
	iState_CP							: INT;							//Variable for the Statemachine to compare
	byStateCH1		AT%I*				: BYTE;							//State Byte from Channel 1 (L1) 
	byCntrCH1		AT%Q*				: BYTE;							//Control Byte from Channel 1 (L1) 
	iDataInCH1		AT%I*				: INT;							//Input Data from Channel 1 (L1) 
	byStateCH2		AT%I*				: BYTE;							//State Byte from Channel 1 (L2) 
	byCntrCH2		AT%Q*				: BYTE;							//Control Byte from Channel 1 (L2) 
	iDataInCH2		AT%I*				: INT;							//Input Data from Channel 1 (L2) 
	byStateCH3		AT%I*				: BYTE;							//State Byte from Channel 1 (L3) 
	byCntrCH3		AT%Q*				: BYTE;							//Control Byte from Channel 1 (L3) 
	iDataInCH3		AT%I*				: INT;							//Input Data from Channel 1 (L3) 
END_VAR

//Creator : Kai Ebensperger
//Company : Lynus AG
//Date : 04.10.2021
//Version : 1.0.0.0

//With this function is possible to read out all Information from a KL3403
//This Function support only the Simple Process Image and the Ratio in the Terminal register must be Set allways to 1.

(*--------------------------------------------------------------------Limits------------------------------------------------------------------------------*)

uiCurrentTransformerRatioL1 := LIMIT(0,uiCurrentTransformerRatioL1,3000);
	uiCurrentTransformerRatioL2 := LIMIT(0,uiCurrentTransformerRatioL2,3000);
		uiCurrentTransformerRatioL3 := LIMIT(0,uiCurrentTransformerRatioL3,3000);
rResolutionCurrent := LIMIT(0,rResolutionCurrent,1);
	rResolutionPower := LIMIT(0,rResolutionPower,1);	
		rResolutionEnergy := LIMIT(0,rResolutionEnergy,1);

(*--------------------------------------------------------------------Errro-Warning------------------------------------------------------------------------------*)		

//Channel 1 (L1)
IF byStateCH1.6 OR NOT timActive.Q OR byStateCH1.7 OR bErrorTimeOut THEN stDataL1.byErrorWarning := 2; ELSE stDataL1.byErrorWarning := 0; END_IF
//Channel 2 (L2)
IF byStateCH2.6 OR NOT timActive.Q OR byStateCH2.7 OR bErrorTimeOut THEN stDataL2.byErrorWarning := 2; ELSE stDataL2.byErrorWarning := 0; END_IF
//Channel 3 (L3)
IF byStateCH3.6 OR NOT timActive.Q OR byStateCH3.7 OR bErrorTimeOut THEN stDataL3.byErrorWarning := 2; ELSE stDataL3.byErrorWarning := 0; END_IF

(*--------------------------------------------------------------------Activate Process data mode------------------------------------------------------------------------------*)		

byCntrCH1.7 := FALSE; byCntrCH1.6 := FALSE;
byCntrCH2.7 := FALSE; byCntrCH2.6 := FALSE;
byCntrCH3.7 := FALSE; byCntrCH3.6 := FALSE;
		
(*--------------------------------------------------------------------Logic part------------------------------------------------------------------------------*)

//Activate the Statemachine when the K-bus is ready
timActive(IN:= uiKBusState_IN = 0, PT:= T#500MS, Q=> , ET=> );
	IF timActive.Q AND iState = 0 THEN iState := 1; END_IF

//Timeout
IF iState > 0 AND iState = iState_CP THEN timTimeout.IN := TRUE; ELSE timTimeout.IN := FALSE; END_IF 
	timTimeout(IN:= , PT:= T#5S, Q=> , ET=> );
	
//State machine
CASE iState OF
	
	1://Set Control Byte for Current
		iState_CP := iState;
	
		//Bin 0000
		byCntrCH1.0 := FALSE; byCntrCH1.1 := FALSE; byCntrCH1.2 := FALSE; byCntrCH1.3 := FALSE;
		byCntrCH2.0 := FALSE; byCntrCH2.1 := FALSE; byCntrCH2.2 := FALSE; byCntrCH2.3 := FALSE;
		byCntrCH3.0 := FALSE; byCntrCH3.1 := FALSE; byCntrCH3.2 := FALSE; byCntrCH3.3 := FALSE;

		//Next Step
		iState := 2;
			
		//Timout Error
		IF timTimeout.Q THEN iState := 300; END_IF	
			
	2://Check Status byte for Current and wirte to the Output Structure
		iState_CP := iState;
			
		//Channel 1 (L1)		
		IF NOT byStateCH1.0 AND NOT byStateCH1.1 AND NOT byStateCH1.2 AND NOT byStateCH1.3 THEN
  			stDataL1.rCurrent := INT_TO_REAL(iDataInCH1) * rResolutionCurrent * uiCurrentTransformerRatioL1;
				arrDataOk[1] := TRUE;
		END_IF 
		//Channel 2 (L2)		
		IF NOT byStateCH2.0 AND NOT byStateCH2.1 AND NOT byStateCH2.2 AND NOT byStateCH2.3 THEN
  			stDataL2.rCurrent := INT_TO_REAL(iDataInCH2) * rResolutionCurrent * uiCurrentTransformerRatioL2;
				arrDataOk[2] := TRUE;
		END_IF 
		//Channel 3 (L3)		
		IF NOT byStateCH3.0 AND NOT byStateCH3.1 AND NOT byStateCH3.2 AND NOT byStateCH3.3 THEN
  			stDataL3.rCurrent := INT_TO_REAL(iDataInCH3) * rResolutionCurrent * uiCurrentTransformerRatioL3;
				arrDataOk[3] := TRUE;
		END_IF 	
		
		//Next Step and prepear controll Byte
		IF arrDataOk[1] AND arrDataOk[2] AND arrDataOk[3] THEN 
			arrDataOk[1] := FALSE; arrDataOk[2] := FALSE; arrDataOk[3] := FALSE;
				//Bin 0001
				byCntrCH1.0 := TRUE; byCntrCH1.1 := FALSE; byCntrCH1.2 := FALSE; byCntrCH1.3 := FALSE;
				byCntrCH2.0 := TRUE; byCntrCH2.1 := FALSE; byCntrCH2.2 := FALSE; byCntrCH2.3 := FALSE;
				byCntrCH3.0 := TRUE; byCntrCH3.1 := FALSE; byCntrCH3.2 := FALSE; byCntrCH3.3 := FALSE;	
					iState := 3; 
		END_IF
		
		//Timout Error
		IF timTimeout.Q THEN iState := 300; END_IF	
		
	3://Check Status byte for Voltage and wirte to the Output Structure
		iState_CP := iState;
			
		//Channel 1 (L1)		
		IF byStateCH1.0 AND NOT byStateCH1.1 AND NOT byStateCH1.2 AND NOT byStateCH1.3 THEN
  			stDataL1.rVoltage := INT_TO_REAL(iDataInCH1) * 0.1;
				arrDataOk[1] := TRUE;
		END_IF 
		//Channel 2 (L2)		
		IF byStateCH2.0 AND NOT byStateCH2.1 AND NOT byStateCH2.2 AND NOT byStateCH2.3 THEN
  			stDataL2.rVoltage := INT_TO_REAL(iDataInCH2) * 0.1;
				arrDataOk[2] := TRUE;
		END_IF 
		//Channel 3 (L3)		
		IF byStateCH3.0 AND NOT byStateCH3.1 AND NOT byStateCH3.2 AND NOT byStateCH3.3 THEN
  			stDataL3.rVoltage := INT_TO_REAL(iDataInCH3) * 0.1;
				arrDataOk[3] := TRUE;
		END_IF 	
		
		//Next Step and prepear controll Byte
		IF arrDataOk[1] AND arrDataOk[2] AND arrDataOk[3] THEN 
			arrDataOk[1] := FALSE; arrDataOk[2] := FALSE; arrDataOk[3] := FALSE;
				//Bin 0010
				byCntrCH1.0 := FALSE; byCntrCH1.1 := TRUE; byCntrCH1.2 := FALSE; byCntrCH1.3 := FALSE;
				byCntrCH2.0 := FALSE; byCntrCH2.1 := TRUE; byCntrCH2.2 := FALSE; byCntrCH2.3 := FALSE;
				byCntrCH3.0 := FALSE; byCntrCH3.1 := TRUE; byCntrCH3.2 := FALSE; byCntrCH3.3 := FALSE;	
					iState := 4; 
		END_IF
		
		//Timout Error
		IF timTimeout.Q THEN iState := 300; END_IF		
	
	4://Check Status byte for Power and wirte to the Output Structure
		iState_CP := iState;
			
		//Channel 1 (L1)		
		IF NOT byStateCH1.0 AND byStateCH1.1 AND NOT byStateCH1.2 AND NOT byStateCH1.3 THEN
  			stDataL1.rPower := INT_TO_REAL(iDataInCH1) * rResolutionPower * uiCurrentTransformerRatioL1;
				arrDataOk[1] := TRUE;
		END_IF 
		//Channel 2 (L2)		
		IF NOT byStateCH2.0 AND byStateCH2.1 AND NOT byStateCH2.2 AND NOT byStateCH2.3 THEN
  			stDataL2.rPower := INT_TO_REAL(iDataInCH2) * rResolutionPower * uiCurrentTransformerRatioL2;
				arrDataOk[2] := TRUE;
		END_IF 
		//Channel 3 (L3)		
		IF NOT byStateCH3.0 AND byStateCH3.1 AND NOT byStateCH3.2 AND NOT byStateCH3.3 THEN
  			stDataL3.rPower := INT_TO_REAL(iDataInCH3) * rResolutionPower * uiCurrentTransformerRatioL3;
				arrDataOk[3] := TRUE;
		END_IF 	
		
		//Next Step and prepear controll Byte
		IF arrDataOk[1] AND arrDataOk[2] AND arrDataOk[3] THEN 
			arrDataOk[1] := FALSE; arrDataOk[2] := FALSE; arrDataOk[3] := FALSE;
				//Bin 0011
				byCntrCH1.0 := TRUE; byCntrCH1.1 := TRUE; byCntrCH1.2 := FALSE; byCntrCH1.3 := FALSE;
				byCntrCH2.0 := TRUE; byCntrCH2.1 := TRUE; byCntrCH2.2 := FALSE; byCntrCH2.3 := FALSE;
				byCntrCH3.0 := TRUE; byCntrCH3.1 := TRUE; byCntrCH3.2 := FALSE; byCntrCH3.3 := FALSE;	
					iState := 5; 
		END_IF
		
		//Timout Error
		IF timTimeout.Q THEN iState := 300; END_IF	
	
	5://Check Status byte for Power factor and wirte to the Output Structure
		iState_CP := iState;
			
		//Channel 1 (L1)		
		IF byStateCH1.0 AND byStateCH1.1 AND NOT byStateCH1.2 AND NOT byStateCH1.3 THEN
  			stDataL1.rPowerfactor := INT_TO_REAL(iDataInCH1) * 0.01;
				arrDataOk[1] := TRUE;
		END_IF 
		//Channel 2 (L2)		
		IF byStateCH2.0 AND byStateCH2.1 AND NOT byStateCH2.2 AND NOT byStateCH2.3 THEN
  			stDataL2.rPowerfactor := INT_TO_REAL(iDataInCH2) * 0.01;
				arrDataOk[2] := TRUE;
		END_IF 
		//Channel 3 (L3)		
		IF byStateCH3.0 AND byStateCH3.1 AND NOT byStateCH3.2 AND NOT byStateCH3.3 THEN
  			stDataL3.rPowerfactor := INT_TO_REAL(iDataInCH3) * 0.01;
				arrDataOk[3] := TRUE;
		END_IF 	
		
		//Next Step and prepear controll Byte
		IF arrDataOk[1] AND arrDataOk[2] AND arrDataOk[3] THEN 
			arrDataOk[1] := FALSE; arrDataOk[2] := FALSE; arrDataOk[3] := FALSE;
				//Bin 0100
				byCntrCH1.0 := FALSE; byCntrCH1.1 := FALSE; byCntrCH1.2 := TRUE; byCntrCH1.3 := FALSE;
				byCntrCH2.0 := FALSE; byCntrCH2.1 := FALSE; byCntrCH2.2 := TRUE; byCntrCH2.3 := FALSE;
				byCntrCH3.0 := FALSE; byCntrCH3.1 := FALSE; byCntrCH3.2 := TRUE; byCntrCH3.3 := FALSE;	
					iState := 6; 
		END_IF
		
		//Timout Error
		IF timTimeout.Q THEN iState := 300; END_IF		
		
	6://Check Status byte for Energy and wirte to the Output Structure
		iState_CP := iState;
			
		//Channel 1 (L1)		
		IF NOT byStateCH1.0 AND NOT byStateCH1.1 AND byStateCH1.2 AND NOT byStateCH1.3 THEN
  			stDataL1.rEnergy := INT_TO_REAL(iDataInCH1) * rResolutionEnergy * uiCurrentTransformerRatioL1;
				arrDataOk[1] := TRUE;
		END_IF 
		//Channel 2 (L2)		
		IF NOT byStateCH2.0 AND NOT byStateCH2.1 AND byStateCH2.2 AND NOT byStateCH2.3 THEN
  			stDataL2.rEnergy := INT_TO_REAL(iDataInCH2) * rResolutionEnergy * uiCurrentTransformerRatioL2;
				arrDataOk[2] := TRUE;
		END_IF 
		//Channel 3 (L3)		
		IF NOT byStateCH3.0 AND NOT byStateCH3.1 AND byStateCH3.2 AND NOT byStateCH3.3 THEN
  			stDataL3.rEnergy := INT_TO_REAL(iDataInCH3) * rResolutionEnergy * uiCurrentTransformerRatioL3;
				arrDataOk[3] := TRUE;
		END_IF 	
		
		//Next Step and prepear controll Byte
		IF arrDataOk[1] AND arrDataOk[2] AND arrDataOk[3] THEN 
			arrDataOk[1] := FALSE; arrDataOk[2] := FALSE; arrDataOk[3] := FALSE;
				//Bin 0101
				byCntrCH1.0 := TRUE; byCntrCH1.1 := FALSE; byCntrCH1.2 := TRUE; byCntrCH1.3 := FALSE;
				byCntrCH2.0 := TRUE; byCntrCH2.1 := FALSE; byCntrCH2.2 := TRUE; byCntrCH2.3 := FALSE;
				byCntrCH3.0 := TRUE; byCntrCH3.1 := FALSE; byCntrCH3.2 := TRUE; byCntrCH3.3 := FALSE;	
					iState := 7; 
		END_IF
		
		//Timout Error
		IF timTimeout.Q THEN iState := 300; END_IF	
	
	7://Check Status byte for Peak Value current and wirte to the Output Structure
		iState_CP := iState;
			
		//Channel 1 (L1)		
		IF byStateCH1.0 AND NOT byStateCH1.1 AND byStateCH1.2 AND NOT byStateCH1.3 THEN
  			stDataL1.rPeakValueCurrent := INT_TO_REAL(iDataInCH1) * rResolutionCurrent * uiCurrentTransformerRatioL1;
				arrDataOk[1] := TRUE;
		END_IF 
		//Channel 2 (L2)		
		IF byStateCH2.0 AND NOT byStateCH2.1 AND byStateCH2.2 AND NOT byStateCH2.3 THEN
  			stDataL2.rPeakValueCurrent := INT_TO_REAL(iDataInCH2) * rResolutionCurrent * uiCurrentTransformerRatioL2;
				arrDataOk[2] := TRUE;
		END_IF 
		//Channel 3 (L3)		
		IF byStateCH3.0 AND NOT byStateCH3.1 AND byStateCH3.2 AND NOT byStateCH3.3 THEN
  			stDataL3.rPeakValueCurrent := INT_TO_REAL(iDataInCH3) * rResolutionCurrent * uiCurrentTransformerRatioL3;
				arrDataOk[3] := TRUE;
		END_IF 	
		
		//Next Step and prepear controll Byte
		IF arrDataOk[1] AND arrDataOk[2] AND arrDataOk[3] THEN 
			arrDataOk[1] := FALSE; arrDataOk[2] := FALSE; arrDataOk[3] := FALSE;
				//Bin 0110
				byCntrCH1.0 := FALSE; byCntrCH1.1 := TRUE; byCntrCH1.2 := TRUE; byCntrCH1.3 := FALSE;
				byCntrCH2.0 := FALSE; byCntrCH2.1 := TRUE; byCntrCH2.2 := TRUE; byCntrCH2.3 := FALSE;
				byCntrCH3.0 := FALSE; byCntrCH3.1 := TRUE; byCntrCH3.2 := TRUE; byCntrCH3.3 := FALSE;	
					iState := 8; 
		END_IF
		
		//Timout Error
		IF timTimeout.Q THEN iState := 300; END_IF
	
	8://Check Status byte for Peak Value voltage and wirte to the Output Structure
		iState_CP := iState;
			
		//Channel 1 (L1)		
		IF NOT byStateCH1.0 AND byStateCH1.1 AND byStateCH1.2 AND NOT byStateCH1.3 THEN
  			stDataL1.rPeakValueVoltage := INT_TO_REAL(iDataInCH1) * 0.1;
				arrDataOk[1] := TRUE;
		END_IF 
		//Channel 2 (L2)		
		IF NOT byStateCH2.0 AND byStateCH2.1 AND byStateCH2.2 AND NOT byStateCH2.3 THEN
  			stDataL2.rPeakValueVoltage := INT_TO_REAL(iDataInCH2) * 0.1;
				arrDataOk[2] := TRUE;
		END_IF 
		//Channel 3 (L3)		
		IF NOT byStateCH3.0 AND byStateCH3.1 AND byStateCH3.2 AND NOT byStateCH3.3 THEN
  			stDataL3.rPeakValueVoltage := INT_TO_REAL(iDataInCH3) * 0.1;
				arrDataOk[3] := TRUE;
		END_IF 	
		
		//Next Step and prepear controll Byte
		IF arrDataOk[1] AND arrDataOk[2] AND arrDataOk[3] THEN 
			arrDataOk[1] := FALSE; arrDataOk[2] := FALSE; arrDataOk[3] := FALSE;
				//Bin 0111
				byCntrCH1.0 := TRUE; byCntrCH1.1 := TRUE; byCntrCH1.2 := TRUE; byCntrCH1.3 := FALSE;
				byCntrCH2.0 := TRUE; byCntrCH2.1 := TRUE; byCntrCH2.2 := TRUE; byCntrCH2.3 := FALSE;
				byCntrCH3.0 := TRUE; byCntrCH3.1 := TRUE; byCntrCH3.2 := TRUE; byCntrCH3.3 := FALSE;	
					iState := 9; 
		END_IF
		
		//Timout Error
		IF timTimeout.Q THEN iState := 300; END_IF	
		
	9://Check Status byte for Peak Value power and wirte to the Output Structure
		iState_CP := iState;
			
		//Channel 1 (L1)		
		IF byStateCH1.0 AND byStateCH1.1 AND byStateCH1.2 AND NOT byStateCH1.3 THEN
  			stDataL1.rPeakValuePower := INT_TO_REAL(iDataInCH1) * rResolutionPower * uiCurrentTransformerRatioL1;
				arrDataOk[1] := TRUE;
		END_IF 
		//Channel 2 (L2)		
		IF byStateCH2.0 AND byStateCH2.1 AND byStateCH2.2 AND NOT byStateCH2.3 THEN
  			stDataL2.rPeakValuePower := INT_TO_REAL(iDataInCH2) * rResolutionPower * uiCurrentTransformerRatioL2;
				arrDataOk[2] := TRUE;
		END_IF 
		//Channel 3 (L3)		
		IF byStateCH3.0 AND byStateCH3.1 AND byStateCH3.2 AND NOT byStateCH3.3 THEN
  			stDataL3.rPeakValuePower := INT_TO_REAL(iDataInCH3) * rResolutionPower * uiCurrentTransformerRatioL3;
				arrDataOk[3] := TRUE;
		END_IF 	
		
		//Next Step and prepear controll Byte
		IF arrDataOk[1] AND arrDataOk[2] AND arrDataOk[3] THEN 
			arrDataOk[1] := FALSE; arrDataOk[2] := FALSE; arrDataOk[3] := FALSE;
				//Bin 1000
				byCntrCH1.0 := FALSE; byCntrCH1.1 := FALSE; byCntrCH1.2 := FALSE; byCntrCH1.3 := TRUE;
				byCntrCH2.0 := FALSE; byCntrCH2.1 := FALSE; byCntrCH2.2 := FALSE; byCntrCH2.3 := TRUE;
				byCntrCH3.0 := FALSE; byCntrCH3.1 := FALSE; byCntrCH3.2 := FALSE; byCntrCH3.3 := TRUE;	
					iState := 10; 
		END_IF
		
		//Timout Error
		IF timTimeout.Q THEN iState := 300; END_IF	
	
	10://Check Status byte for Frequency and wirte to the Output Structure
		iState_CP := iState;
			
		//Channel 1 (L1)		
		IF NOT byStateCH1.0 AND NOT byStateCH1.1 AND NOT byStateCH1.2 AND byStateCH1.3 THEN
  			stDataL1.rFrequency := INT_TO_REAL(iDataInCH1) * 0.1;
				arrDataOk[1] := TRUE;
		END_IF 
		//Channel 2 (L2)		
		IF NOT byStateCH2.0 AND NOT byStateCH2.1 AND NOT byStateCH2.2 AND byStateCH2.3 THEN
  			stDataL2.rFrequency := INT_TO_REAL(iDataInCH2) * 0.1;
				arrDataOk[2] := TRUE;
		END_IF 
		//Channel 3 (L3)		
		IF NOT byStateCH3.0 AND NOT byStateCH3.1 AND NOT byStateCH3.2 AND byStateCH3.3 THEN
  			stDataL3.rFrequency := INT_TO_REAL(iDataInCH3) * 0.1;
				arrDataOk[3] := TRUE;
		END_IF 	
		
		//Next Step and prepear controll Byte
		IF arrDataOk[1] AND arrDataOk[2] AND arrDataOk[3] THEN 
			arrDataOk[1] := FALSE; arrDataOk[2] := FALSE; arrDataOk[3] := FALSE;
				//Bin 1001
				byCntrCH1.0 := TRUE; byCntrCH1.1 := FALSE; byCntrCH1.2 := FALSE; byCntrCH1.3 := TRUE;
				byCntrCH2.0 := TRUE; byCntrCH2.1 := FALSE; byCntrCH2.2 := FALSE; byCntrCH2.3 := TRUE;
				byCntrCH3.0 := TRUE; byCntrCH3.1 := FALSE; byCntrCH3.2 := FALSE; byCntrCH3.3 := TRUE;	
					iState := 11; 
		END_IF
		
		//Timout Error
		IF timTimeout.Q THEN iState := 300; END_IF
	
	11://Check Status byte for Min value current and wirte to the Output Structure
		iState_CP := iState;
			
		//Channel 1 (L1)		
		IF byStateCH1.0 AND NOT byStateCH1.1 AND NOT byStateCH1.2 AND byStateCH1.3 THEN
  			stDataL1.rMinValueCurrent := INT_TO_REAL(iDataInCH1) * rResolutionCurrent * uiCurrentTransformerRatioL1;
				arrDataOk[1] := TRUE;
		END_IF 
		//Channel 2 (L2)		
		IF byStateCH2.0 AND NOT byStateCH2.1 AND NOT byStateCH2.2 AND byStateCH2.3 THEN
  			stDataL2.rMinValueCurrent := INT_TO_REAL(iDataInCH2) * rResolutionCurrent * uiCurrentTransformerRatioL2;
				arrDataOk[2] := TRUE;
		END_IF 
		//Channel 3 (L3)		
		IF byStateCH3.0 AND NOT byStateCH3.1 AND NOT byStateCH3.2 AND byStateCH3.3 THEN
  			stDataL3.rMinValueCurrent := INT_TO_REAL(iDataInCH3) * rResolutionCurrent * uiCurrentTransformerRatioL3;
				arrDataOk[3] := TRUE;
		END_IF 	
		
		//Next Step and prepear controll Byte
		IF arrDataOk[1] AND arrDataOk[2] AND arrDataOk[3] THEN 
			arrDataOk[1] := FALSE; arrDataOk[2] := FALSE; arrDataOk[3] := FALSE;
				//Bin 1010
				byCntrCH1.0 := FALSE; byCntrCH1.1 := TRUE; byCntrCH1.2 := FALSE; byCntrCH1.3 := TRUE;
				byCntrCH2.0 := FALSE; byCntrCH2.1 := TRUE; byCntrCH2.2 := FALSE; byCntrCH2.3 := TRUE;
				byCntrCH3.0 := FALSE; byCntrCH3.1 := TRUE; byCntrCH3.2 := FALSE; byCntrCH3.3 := TRUE;	
					iState := 12; 
		END_IF
		
		//Timout Error
		IF timTimeout.Q THEN iState := 300; END_IF	
		
	12://Check Status byte for Min value voltage and wirte to the Output Structure
		iState_CP := iState;
			
		//Channel 1 (L1)		
		IF NOT byStateCH1.0 AND byStateCH1.1 AND NOT byStateCH1.2 AND byStateCH1.3 THEN
  			stDataL1.rMinValueVoltage := INT_TO_REAL(iDataInCH1) * 0.1;
				arrDataOk[1] := TRUE;
		END_IF 
		//Channel 2 (L2)		
		IF NOT byStateCH2.0 AND byStateCH2.1 AND NOT byStateCH2.2 AND byStateCH2.3 THEN
  			stDataL2.rMinValueVoltage := INT_TO_REAL(iDataInCH2) * 0.1;
				arrDataOk[2] := TRUE;
		END_IF 
		//Channel 3 (L3)		
		IF NOT byStateCH3.0 AND byStateCH3.1 AND NOT byStateCH3.2 AND byStateCH3.3 THEN
  			stDataL3.rMinValueVoltage := INT_TO_REAL(iDataInCH3) * 0.1;
				arrDataOk[3] := TRUE;
		END_IF 	
		
		//Next Step and prepear controll Byte
		IF arrDataOk[1] AND arrDataOk[2] AND arrDataOk[3] THEN 
			arrDataOk[1] := FALSE; arrDataOk[2] := FALSE; arrDataOk[3] := FALSE;
				//Bin 1011
				byCntrCH1.0 := TRUE; byCntrCH1.1 := TRUE; byCntrCH1.2 := FALSE; byCntrCH1.3 := TRUE;
				byCntrCH2.0 := TRUE; byCntrCH2.1 := TRUE; byCntrCH2.2 := FALSE; byCntrCH2.3 := TRUE;
				byCntrCH3.0 := TRUE; byCntrCH3.1 := TRUE; byCntrCH3.2 := FALSE; byCntrCH3.3 := TRUE;	
					iState := 13; 
		END_IF
		
		//Timout Error
		IF timTimeout.Q THEN iState := 300; END_IF	
		
	13://Check Status byte for Min value power and wirte to the Output Structure
		iState_CP := iState;
			
		//Channel 1 (L1)		
		IF byStateCH1.0 AND byStateCH1.1 AND NOT byStateCH1.2 AND byStateCH1.3 THEN
  			stDataL1.rMinValuePower := INT_TO_REAL(iDataInCH1) * rResolutionPower * uiCurrentTransformerRatioL1;
				arrDataOk[1] := TRUE;
		END_IF 
		//Channel 2 (L2)		
		IF byStateCH2.0 AND byStateCH2.1 AND NOT byStateCH2.2 AND byStateCH2.3 THEN
  			stDataL2.rMinValuePower := INT_TO_REAL(iDataInCH2) * rResolutionPower * uiCurrentTransformerRatioL2;
				arrDataOk[2] := TRUE;
		END_IF 
		//Channel 3 (L3)		
		IF byStateCH3.0 AND byStateCH3.1 AND NOT byStateCH3.2 AND byStateCH3.3 THEN
  			stDataL3.rMinValuePower := INT_TO_REAL(iDataInCH3) * rResolutionPower * uiCurrentTransformerRatioL3;
				arrDataOk[3] := TRUE;
		END_IF 	
		
		//Next Step and prepear controll Byte
		IF arrDataOk[1] AND arrDataOk[2] AND arrDataOk[3] THEN 
			arrDataOk[1] := FALSE; arrDataOk[2] := FALSE; arrDataOk[3] := FALSE;
				//Start from New	
				iState := 1;
					bErrorTimeOut := FALSE; 
		END_IF
		
		//Timout Error
		IF timTimeout.Q THEN iState := 300; END_IF	
		
	300://Error
		bErrorTimeOut := TRUE;
		
		//Start from new with the Statemachine
		iState := 1;

END_CASE

END_FUNCTION_BLOCK

// ---- Energy/FBs Internal/Beckhoff/FB_XL1XXX_DI.TcPOU
{attribute 'conditionalshow'}
FUNCTION_BLOCK FB_XL1XXX_DI
VAR_INPUT
	{attribute 'hide'}
	bInvers							: BOOL;				//Invert the input signal
END_VAR
VAR_OUTPUT
	{attribute 'hide'}
	bSignal							: BOOL;				//Signal from the terminal
END_VAR
VAR
	bDataIn					AT%I*	: BOOL;				//Input data from the termianl 
END_VAR

//Creator : Kai Ebensperger
//Company : Lynus AG
//Date : 02.06.2021
//Version : 1.0.0.0

//With this fuction block its possible to read in a digital signal from a Beckhoff Digital Input terminal
//Here we have the possibility to invert the input signal

IF NOT bInvers THEN 
	bSignal := bDataIn;
ELSE
	bSignal := NOT bDataIn;
END_IF

END_FUNCTION_BLOCK

// ---- Energy/FBs Internal/Beckhoff/FB_XL2XXX_DO.TcPOU
{attribute 'conditionalshow'}
FUNCTION_BLOCK FB_XL2XXX_DO
VAR_INPUT
	{attribute 'hide'}
	bInvers							: BOOL;				//Invert the output signal
	{attribute 'hide'}
	bSignal							: BOOL;				//Signal to send to the terminal
END_VAR
VAR_OUTPUT
END_VAR
VAR
	bDataOut		AT%Q*			: BOOL;				//Output Data for the terminal
END_VAR

//Creator : Kai Ebensperger
//Company : Lynus AG
//Date : 02.06.2021
//Version : 1.0.0.0

//With this function block its possible to send a digital signal from the plc to a digital output terminal from Beckhoff
//We have also the possibility to invert the output signal
	
IF NOT bInvers THEN
	bDataOut := bSignal;
ELSE
	bDataOut := NOT bSignal;
END_IF

END_FUNCTION_BLOCK

// ---- Energy/FBs Internal/Beckhoff/FB_XL3XXX_AI.TcPOU
{attribute 'conditionalshow'}
FUNCTION_BLOCK FB_XL3XXX_AI
VAR_INPUT
	{attribute 'hide'}
	rXMinTerminalValue		: REAL;				//Min value from the Terminal for scalling
	{attribute 'hide'}
	rYMinOutputSignal		: REAL;				//Min value from the new output signal for scalling
	{attribute 'hide'}
	rXMaxTerminalValue		: REAL;				//Max value from the Terminal for scalling
	{attribute 'hide'}
	rYMaxOutputSignal		: REAL;				//Max value from the new output signal for scalling
END_VAR
VAR_OUTPUT
	usiState	AT%I*		: USINT;			//State from the terminal
	{attribute 'hide'}
	rSignal					: REAL;				//New output signal
END_VAR	
VAR
	iDataIn		AT%I*		: INT;				//Raw Input value from the terminal
END_VAR

//Creator : Kai Ebensperger
//Company : Lynus AG
//Date : 02.06.2021
//Version : 1.0.0.0

//With this function block its possible to read in a analog signal from a beckhoff analog input terminal and convert in the right size. 32767 to 10 for example

(*---------------------------------------------------------------Check the limits of the inputs-------------------------------------------------------------------------------*)

rXMinTerminalValue := LIMIT(0,rXMinTerminalValue,32767);
	rXMaxTerminalValue := LIMIT(0,rXMaxTerminalValue,32767);	

(*----------------------------------------------------------------------Scalling----------------------------------------------------------------------------------------------*)

rSignal := F_Scalvalue(x:= INT_TO_REAL(iDataIn), x1:= rXMinTerminalValue, y1:= rYMinOutputSignal, x2:= rXMaxTerminalValue, y2:= rYMaxOutputSignal,);

END_FUNCTION_BLOCK

// ---- Energy/FBs Internal/Beckhoff/FB_XL4XXX_AO.TcPOU
{attribute 'conditionalshow'}
FUNCTION_BLOCK FB_XL4XXX_AO
VAR_INPUT
	{attribute 'hide'}
	rYMinTerminalValue		: REAL;				//Min value from the Terminal for scalling
	{attribute 'hide'}
	rXMinInputSignal		: REAL;				//Min value from the new input signal for scalling
	{attribute 'hide'}
	rYMaxTerminalValue		: REAL;				//Max value from the Terminal for scalling
	{attribute 'hide'}
	rXMaxInputSignal		: REAL;				//Max value from the new input signal for scalling
	{attribute 'hide'}
	rSignal					: REAL;				//New Input signal
END_VAR
VAR_OUTPUT
	usiState	AT%I*		: USINT;			//State from the terminal
END_VAR
VAR
	iDataOut	AT%Q*		: INT;				//Raw output value for the terminal
	{attribute 'hide'}
	rValue					: REAL;				//Internal value to check
END_VAR

//Creator : Kai Ebensperger
//Company : Lynus AG
//Date : 02.06.2021
//Version : 1.0.0.0

//With this function block its possible to write out a analog signal to a beckhoff analog output terminal and convert before in the right size. 10 to 32767 for example

(*---------------------------------------------------------------Check the limits of the inputs-------------------------------------------------------------------------------*)

rYMinTerminalValue := LIMIT(0,rYMinTerminalValue,32767);
	rYMaxTerminalValue := LIMIT(0,rYMaxTerminalValue,32767);
	
(*----------------------------------------------------------------------Scalling----------------------------------------------------------------------------------------------*)

rValue := F_Scalvalue(x:= rSignal, x1:= rXMinInputSignal, y1:= rYMinTerminalValue, x2:= rXMaxInputSignal, y2:= rYMaxTerminalValue,);
	rValue := LIMIT(0,rValue,32767);
		iDataOut := REAL_TO_INT(rValue);

END_FUNCTION_BLOCK

// ---- Energy/FBs Internal/Controller/FB_PID.TcPOU
{attribute 'hide_all_locals'}
{attribute 'conditionalshow'}
FUNCTION_BLOCK FB_PID
VAR_INPUT
	{attribute 'hide'}
	bEnable					: BOOL;						//Enable the regulation
	{attribute 'hide'}
	rSetpoint				: REAL;						//Setpoint to which the controller controls
	{attribute 'hide'}
	udiIValue				: UDINT;					//Reset time
	{attribute 'hide'}
	udiDValue				: UDINT;					//Lead time
	{attribute 'hide'}
	udiDamping				: UDINT;					//Damping
	{attribute 'hide'}
	rPValue					: REAL;						//Controller gain
	{attribute 'hide'}
	rMaxValue				: REAL;						//Max Value from the output of the controller
	{attribute 'hide'}
	rMinValue				: REAL;						//Min Value from the output of the controller
	{attribute 'hide'}
	rNeutralZone			: REAL;						//If the value of the control deviation is smaller than half of lrNeutralZone, the control signal remains the same
	{attribute 'hide'}
	bDirection				: BOOL;						//Direction from the controller
	{attribute 'hide'}
	rActualValue			: REAL;						//Current value that the controller tries to adapt to the setpoint and to regulate
END_VAR
VAR_OUTPUT
	{attribute 'hide'}
	rQController			: REAL;						//Controller output
END_VAR
VAR
	PIDController			: FB_BA_PIDCtrl;			//PID controller
END_VAR

//Creator : Kai Ebensperger
//Company : Lynus AG
//Date : 19.05.2021
//Version : 1.0.0.0

//This function block represents a classic PID controller that can be set individually.
PIDController(
	bEn:= bEnable, 
	rW:= rSetpoint, 
	rX:= rActualValue, 
	udiOpMode:= 0, 
	bActn:= bDirection, 
	rKp:= rPValue, 
	udiTn_ms:= udiIValue, 
	udiTv_ms:= udiDValue, 
	udiTd_ms:= udiDamping, 
	rYMax:= rMaxValue, 
	rYMin:= rMinValue, 
	rNZ:= rNeutralZone, 
	udiCycCl:= 1, 
	bSync:= , 
	rSync:= , 
	rY=> rQController, 
	rE=> , 
	bARW=> );

END_FUNCTION_BLOCK

// ---- Energy/FBs Internal/Electric CS/FB_ElectricChargingStation.TcPOU
{attribute 'hide_all_locals'}
{attribute 'conditionalshow'}
FUNCTION_BLOCK FB_ElectricChargingStation
VAR_INPUT
	{attribute 'hide'}
	bEnable									: BOOL;									//Enable the Fuctionblock and his logic
	{attribute 'hide'}
	bError									: BOOL;									//Error Input charging station
	{attribute 'hide'}
	bWarning								: BOOL;									//Warning Input charging station
	{attribute 'hide'}
	bEPOIsActive							: BOOL;									//Emergency power operation is active
	{attribute 'hide'}
	bExternalLock							: BOOL;									//External lock (All functions are locked)
	{attribute 'hide'}
	bCarConnected							: BOOL;									//Feedback if the car is connected to the charging station
	{attribute 'hide'}
	bWriteWithDelay							: BOOL;									//Write with Delay the Data to the output (Not al Output Data is writen with Delay)
	{attribute 'hide'}
	bCalculateEnergySession					: BOOL;									//When its true then the Energy Session is calculatet by the diffference of arrEnergySession[] when we have a change. FALSE = Use direct the Input from arrEnergySession[]
	{attribute 'hide'}
	iErrorCode								: INT;									//Error Code from external ECS
	{attribute 'hide'}
	iWarningCode							: INT;									//Warning Code from external ECS
	{attribute 'hide'}							
	dwBatterySOC							: DWORD;								//Actual Battery SOC in %
	{attribute 'hide'}
	lrTotalCounterEnergy_Consumption		: LREAL;								//Total Counter for Energy consumption with unit Wh
	{attribute 'hide'}
	lrTotalCounterEnergy_Production			: LREAL;								//Total Counter for Energy production with unit Wh
	{attribute 'hide'}
	lrCounterEnergyT1_Consumption			: LREAL;								//Total counter for energy Tariff 1 consumption with unit Wh
	{attribute 'hide'}
	lrCounterEnergyT2_Consumption			: LREAL;								//Total counter for energy Tariff 2 consumption with unit Wh
	{attribute 'hide'}
	lrCounterEnergyT1_Production			: LREAL;								//Total counter for energy Tariff 1 production with unit Wh
	{attribute 'hide'}
	lrCounterEnergyT2_Production			: LREAL;								//Total counter for energy Tariff 2 production with unit Wh
	{attribute 'hide'}
	lrTotalPowerECS							: LREAL;								//Input Value from the total power of the charging station with unit W
	{attribute 'hide'}
	rTargetPower							: REAL;									//Target power from 0% to +100%
	{attribute 'hide'}
	rSupplyVoltage							: REAL;									//Supply voltage of the charging station for current calculation
	{attribute 'hide'}
	rMinCurrent								: REAL;									//Min. current that must flow for the charging station to switch on (if the current falls below this value, the car will not accept charging)
	{attribute 'hide'}
	tTimDelayOutput							: TIME := T#5S;							//Delay Time to write some Data to the Output	
	{attribute 'hide'}
	tDelayError								: TIME := T#15S;						//Delay for Error
	{attribute 'hide'}	
	arrSocketMode3StateECS					: ARRAY[1..4] OF STRING(2);				//Mode 3 State Charging Station of each socket (A + E = ECS Ready or free, B1 + B2 + C1 + D1 = Car connected, C2 + D2 = Charging, F = Error)
	{attribute 'hide'}	
	arrSOCCar								: ARRAY[1..4] OF DWORD;					//SOC from the car from each socket. 0 - 100%
	{attribute 'hide'}	
	arrSocketChargingTimeInput				: ARRAY[1..4] OF REAL;					//Past charging time in min from each socket
	{attribute 'hide'}	
	arrSocketEnergySession					: ARRAY[1..4] OF LREAL;					//Input for Energy Session or total Energy Counter of each socket. Look at the Input bCalculateEnergySession. Wh
	{attribute 'hide'}	
	arrSocketPowerECS						: ARRAY[1..4] OF LREAL;					//Input Value from the power of each socket from the charging station with unit W
	{attribute 'hide'}
	stSetupECS								: ST_Setup_ECS;							//Setup charging station
END_VAR
VAR_OUTPUT
	{attribute 'hide'}
	stDataECSOut							: ST_ECS_Output;						//Electric charging station output data
	{attribute 'hide'}
	stDataECSOutDelay						: ST_ECS_Output;						//Electric charging station output data with delay
END_VAR
VAR
	FPEnable								: R_TRIG;								//Internal positive Edge
	FNManualy								: F_TRIG;								//Internal negative edge
	FNEnable								: F_TRIG;								//Internal negative Edge
	timDelayOutputs							: TON;									//Timer to send Data with Delay to the outputs
	timError								: TON;									//Timer to set the error
	timSOCDissable							: TON;									//Delay to dissable the ECS when the battery SOC has reached the value to dissale
	bMinCurrent								: BOOL;									//Current is fallen below min
	rMaxCurrent								: REAL;									//Max current from the charging station
	rPorcentOn								: REAL;									//Porcent value when the charging station switch on
	FPMode3C2								: ARRAY[1..4] OF R_TRIG;				//Internal positive Edge
	FPMode3D2								: ARRAY[1..4] OF R_TRIG;				//Internal positive Edge
	arrEnergySession_Cmp					: ARRAY[1..4] OF LREAL;					//Total Energy Comsumption for calculation of the energy session
END_VAR

//Creator : Kai Ebensperger
//Company : Lynus AG
//Date : 19.05.2021
//Version : 1.0.0.0

//This function block can be used to display the basic logic of a charging station.
//The charging station can either be switched on manually, in which case the power specification is not observed
//Otherwise the switching output of the charging station is set at 100% power setting
//In the power default mode, the SOC of the battery must be between On and Off SOC and must have reached On SOC once
//< Constants.byTargetOffPowerOnOffDevices the output is reset because of the hysteresis
//This FB can be used for charging stations on/off and for those which can be controlled linearly.
//Furthermore, the FB has an external blocking signal which switches off all functions as long as this is active.
//In addition, the FB outputs the power specification in parallel as a current specification. Ratio between power and voltage

(*---------------------------------------------------------------Check the limits of the inputs-------------------------------------------------------------------------------*)

arrSOCCar[1] := LIMIT(0,arrSOCCar[1],100); arrSOCCar[2] := LIMIT(0,arrSOCCar[2],100); arrSOCCar[3] := LIMIT(0,arrSOCCar[3],100); arrSOCCar[4] := LIMIT(0,arrSOCCar[4],100);
	dwBatterySOC := LIMIT(0,dwBatterySOC,100);
		rTargetPower := LIMIT(0,rTargetPower,100);
			stSetupECS.byManualyTargetPower := LIMIT(0,stSetupECS.byManualyTargetPower,100);
				stSetupECS.rMaxPower := LIMIT(0,stSetupECS.rMaxPower,500);
					stSetupECS.byCSMinPower := LIMIT(0,stSetupECS.byCSMinPower,100);	
						arrSocketChargingTimeInput[1] := LIMIT(0,arrSocketChargingTimeInput[1],100000); arrSocketChargingTimeInput[2] := LIMIT(0,arrSocketChargingTimeInput[2],100000); arrSocketChargingTimeInput[3] := LIMIT(0,arrSocketChargingTimeInput[3],100000); arrSocketChargingTimeInput[4] := LIMIT(0,arrSocketChargingTimeInput[4],100000);
							rSupplyVoltage := LIMIT(0,rSupplyVoltage,1000);
							
IF IsFinite(F_LREAL(lrTotalCounterEnergy_Consumption)) THEN lrTotalCounterEnergy_Consumption := LIMIT(0,lrTotalCounterEnergy_Consumption,999999999999999); END_IF
	IF IsFinite(F_LREAL(lrTotalCounterEnergy_Production)) THEN lrTotalCounterEnergy_Production := LIMIT(0,lrTotalCounterEnergy_Production,999999999999999); END_IF
		IF IsFinite(F_LREAL(lrCounterEnergyT1_Consumption)) THEN lrCounterEnergyT1_Consumption := LIMIT(0,lrCounterEnergyT1_Consumption,999999999999999); END_IF
			IF IsFinite(F_LREAL(lrCounterEnergyT2_Consumption)) THEN lrCounterEnergyT2_Consumption := LIMIT(0,lrCounterEnergyT2_Consumption,999999999999999); END_IF
				IF IsFinite(F_LREAL(lrCounterEnergyT1_Production)) THEN lrCounterEnergyT1_Production := LIMIT(0,lrCounterEnergyT1_Production,999999999999999); END_IF
					IF IsFinite(F_LREAL(lrCounterEnergyT2_Production)) THEN lrCounterEnergyT2_Production := LIMIT(0,lrCounterEnergyT2_Production,999999999999999); END_IF
						lrTotalPowerECS := LIMIT(-999999999999999,lrTotalPowerECS,999999999999999);
							arrSocketPowerECS[1] := LIMIT(-999999999999999,arrSocketPowerECS[1],999999999999999);
								arrSocketPowerECS[2] := LIMIT(-999999999999999,arrSocketPowerECS[2],999999999999999);
									arrSocketPowerECS[3] := LIMIT(-999999999999999,arrSocketPowerECS[3],999999999999999);
										arrSocketPowerECS[4] := LIMIT(-999999999999999,arrSocketPowerECS[4],999999999999999);
											IF IsFinite(F_LREAL(arrSocketEnergySession[1])) THEN arrSocketEnergySession[1] := LIMIT(0,arrSocketEnergySession[1],999999999999999); END_IF
												IF IsFinite(F_LREAL(arrSocketEnergySession[2])) THEN arrSocketEnergySession[2] := LIMIT(0,arrSocketEnergySession[2],999999999999999); END_IF
													IF IsFinite(F_LREAL(arrSocketEnergySession[3])) THEN arrSocketEnergySession[3] := LIMIT(0,arrSocketEnergySession[3],999999999999999); END_IF
														IF IsFinite(F_LREAL(arrSocketEnergySession[4])) THEN arrSocketEnergySession[4] := LIMIT(0,arrSocketEnergySession[4],999999999999999); END_IF
					
IF stSetupECS.byDisableSOC > stSetupECS.byEnableSOC THEN stSetupECS.byEnableSOC := stSetupECS.byDisableSOC + 1; END_IF

stSetupECS.byDisableSOC := LIMIT(0,stSetupECS.byDisableSOC,100);
	stSetupECS.byEnableSOC := LIMIT(1,stSetupECS.byEnableSOC,100);

(*---------------------------------------------------------------------------Enable----------------------------------------------------------------------------------*)

stDataECSOut.bEnabled := bEnable;

(*-----------------------------------------------------------------------------Error and Warning----------------------------------------------------------------------------*)

timError(IN:= bError, PT:= tDelayError, Q=> , ET=> );

stDataECSOut.byErrorWarning := 0;
	IF bWarning THEN stDataECSOut.byErrorWarning := 1; END_IF 
	IF timError.Q THEN stDataECSOut.byErrorWarning := 2; END_IF

//Messages and Error Codes
IF bExternalLock THEN stDataECSOut.eMessage := E_Message_ECS.eExternalLockActive;
ELSIF stDataECSOut.byErrorWarning = 1 AND iWarningCode = 0 THEN stDataECSOut.eMessage := E_Message_ECS.eNoConnectionToBackend;
ELSIF stDataECSOut.byErrorWarning = 1 AND iWarningCode = 1 THEN stDataECSOut.eMessage := E_Message_ECS.eWarningECS;
ELSIF stDataECSOut.byErrorWarning = 2 AND iErrorCode = 0 THEN stDataECSOut.eMessage := E_Message_ECS.eErrorECS;
ELSIF stDataECSOut.byErrorWarning = 2 AND iErrorCode = 1 THEN stDataECSOut.eMessage := E_Message_ECS.eTooMuchECS;
ELSE stDataECSOut.eMessage := E_Message_ECS.eNoMessage; 
END_IF

(*----------------------------------------------------------------------------Logic Part------------------------------------------------------------------------------------*)

//Target power
stDataECSOut.rTargetPower := DINT_TO_REAL(REAL_TO_DINT(rTargetPower * 100)) / 100;
IF rTargetPower <= stSetupECS.byCSMinPower THEN stDataECSOut.rTargetPower := BYTE_TO_REAL(stSetupECS.byCSMinPower); END_IF 
IF stSetupECS.bManualyOn THEN stDataECSOut.rTargetPower := BYTE_TO_REAL(stSetupECS.byManualyTargetPower); END_IF  

//When the current is fallen below the minimum then the charging station is switching off
//Calculate the max current for this charging station
IF rSupplyVoltage > 0 THEN
	rMaxCurrent := (stSetupECS.rMaxPower * 1000) / rSupplyVoltage;
ELSE
	rMaxCurrent := 0;
END_IF
	stDataECSOut.rTargetChargeCurrent := F_Scalvalue(x:= stDataECSOut.rTargetPower, x1:= 0, y1:= 0, x2:= 100, y2:= rMaxCurrent); 
	
IF rMaxCurrent = 0 THEN bMinCurrent := TRUE; ELSE bMinCurrent := FALSE; END_IF

//Calculate the porcent value for the min current
IF rMaxCurrent > 0 THEN
	rPorcentOn := (100 * rMinCurrent) / rMaxCurrent;
ELSE
	rPorcentOn := 0;
END_IF

//Timer for SOC Dissable
timSOCDissable(IN:= dwBatterySOC <= stSetupECS.byDisableSOC, PT:= T#30S, Q=> , ET=> );
	
//Switch Off
FNManualy(CLK:= stSetupECS.bManualyOn, Q=> ); 

IF NOT bEnable OR bMinCurrent OR bExternalLock OR stDataECSOut.byErrorWarning = 2 OR stDataECSOut.rTargetPower <= 0 OR timSOCDissable.Q OR (bEPOIsActive AND stSetupECS.bOnEmergPowerOff) OR FNManualy.Q THEN
	stDataECSOut.bOutput := FALSE;
END_IF

//Switch On
IF (bEnable AND NOT bExternalLock AND stDataECSOut.byErrorWarning <> 2 AND NOT bMinCurrent AND NOT bEPOIsActive AND stDataECSOut.rTargetPower > rPorcentOn AND dwBatterySOC >= stSetupECS.byEnableSOC) OR 
	(bEnable AND NOT bExternalLock AND stDataECSOut.byErrorWarning <> 2 AND bEPOIsActive AND NOT bMinCurrent AND NOT stSetupECS.bOnEmergPowerOff AND stDataECSOut.rTargetPower > rPorcentOn AND dwBatterySOC >= stSetupECS.byEnableSOC) OR
		(bEnable AND NOT bExternalLock AND NOT bMinCurrent AND stDataECSOut.byErrorWarning <> 2 AND stSetupECS.bManualyOn AND stDataECSOut.rTargetPower > rPorcentOn) THEN	
			stDataECSOut.bOutput := TRUE;
END_IF 

//Use this Output to switch Charging station on and off without possibility to send a target power value (Not controllable)
IF stDataECSOut.rTargetPower >= 100 AND stDataECSOut.bOutput THEN stDataECSOut.bOutputOnOff := TRUE; END_IF  
IF stDataECSOut.rTargetPower < Constants_Energy.byTargetOffPowerForOnOffDevices OR NOT stDataECSOut.bOutput THEN stDataECSOut.bOutputOnOff := FALSE; END_IF  

IF NOT stDataECSOut.bOutput THEN stDataECSOut.rTargetPower := 0; stDataECSOut.rTargetChargeCurrent := 0; END_IF 

IF stDataECSOut.rTargetChargeCurrent < rMinCurrent AND stDataECSOut.bOutput THEN stDataECSOut.rTargetChargeCurrent := rMinCurrent; END_IF

stDataECSOut.rTargetChargeCurrent := DINT_TO_REAL(REAL_TO_DINT(stDataECSOut.rTargetChargeCurrent * 100)) / 100;

(*------------------------------------------------------------------Power data----------------------------------------------------------------------------------------------*)

IF bEnable THEN
	stDataECSOut.lrTotalPower:= LINT_TO_LREAL(LREAL_TO_LINT((lrTotalPowerECS / 1000) * 100)) / 100;
		IF IsFinite(F_LREAL(lrCounterEnergyT1_Consumption)) THEN stDataECSOut.lrCounterEnergyT1_Consumption := LINT_TO_LREAL(LREAL_TO_LINT((lrCounterEnergyT1_Consumption / 1000) * 100)) / 100; END_IF
			IF IsFinite(F_LREAL(lrCounterEnergyT2_Consumption)) THEN stDataECSOut.lrCounterEnergyT2_Consumption := LINT_TO_LREAL(LREAL_TO_LINT((lrCounterEnergyT2_Consumption / 1000) * 100)) / 100; END_IF
				IF IsFinite(F_LREAL(lrCounterEnergyT1_Production)) THEN stDataECSOut.lrCounterEnergyT1_Production := LINT_TO_LREAL(LREAL_TO_LINT((lrCounterEnergyT1_Production / 1000) * 100)) / 100; END_IF
					IF IsFinite(F_LREAL(lrCounterEnergyT2_Production)) THEN stDataECSOut.lrCounterEnergyT2_Production := LINT_TO_LREAL(LREAL_TO_LINT((lrCounterEnergyT2_Production / 1000) * 100)) / 100; END_IF
						IF IsFinite(F_LREAL(lrTotalCounterEnergy_Consumption)) THEN stDataECSOut.lrTotalCounterEnergy_Consumption := LINT_TO_LREAL(LREAL_TO_LINT((lrTotalCounterEnergy_Consumption / 1000) * 100)) / 100; END_IF
							IF IsFinite(F_LREAL(lrTotalCounterEnergy_Production)) THEN stDataECSOut.lrTotalCounterEnergy_Production := LINT_TO_LREAL(LREAL_TO_LINT((lrTotalCounterEnergy_Production / 1000) * 100)) / 100; END_IF 
				
		IF stDataECSOut.lrTotalPower < 0 THEN
				stDataECSOut.lrTotalPowerProduction := (stDataECSOut.lrTotalPower * - 1);
				stDataECSOut.lrTotalPowerConsumption := 0;
		ELSIF stDataECSOut.lrTotalPower > 0 THEN
				stDataECSOut.lrTotalPowerProduction := 0;
				stDataECSOut.lrTotalPowerConsumption := stDataECSOut.lrTotalPower;
		ELSIF stDataECSOut.lrTotalPower = 0 THEN
				stDataECSOut.lrTotalPowerProduction := 0;
				stDataECSOut.lrTotalPowerConsumption := 0;
		END_IF
		
		//Socket Power
		stDataECSOut.arrSocketPower[1] := LINT_TO_LREAL(LREAL_TO_LINT((arrSocketPowerECS[1] / 1000) * 100)) / 100;
			stDataECSOut.arrSocketPower[2] := LINT_TO_LREAL(LREAL_TO_LINT((arrSocketPowerECS[2] / 1000) * 100)) / 100;
				stDataECSOut.arrSocketPower[3] := LINT_TO_LREAL(LREAL_TO_LINT((arrSocketPowerECS[3] / 1000) * 100)) / 100;
					stDataECSOut.arrSocketPower[4] := LINT_TO_LREAL(LREAL_TO_LINT((arrSocketPowerECS[4] / 1000) * 100)) / 100;
		
ELSE
	stDataECSOut.lrTotalPower := 0;
		stDataECSOut.lrCounterEnergyT1_Consumption := 0;
			stDataECSOut.lrCounterEnergyT2_Consumption := 0;
				stDataECSOut.lrCounterEnergyT1_Production := 0;
					stDataECSOut.lrCounterEnergyT2_Production := 0;
						stDataECSOut.lrTotalPowerProduction := 0;
							stDataECSOut.lrTotalPowerConsumption := 0;	
								stDataECSOut.lrTotalCounterEnergy_Consumption := 0;
									stDataECSOut.lrTotalCounterEnergy_Production := 0;
									
	//Socket
	stDataECSOut.arrSocketPower[1] := 0;
			stDataECSOut.arrSocketPower[2] := 0;
				stDataECSOut.arrSocketPower[3] := 0;
					stDataECSOut.arrSocketPower[4] := 0;
END_IF

//Calcualte Energy from actual Session
FPMode3C2[1](CLK:= arrSocketMode3StateECS[1] = 'C2', Q=> );
	FPMode3D2[1](CLK:= arrSocketMode3StateECS[1] = 'D2', Q=> );
		FPMode3C2[2](CLK:= arrSocketMode3StateECS[2] = 'C2', Q=> );
			FPMode3D2[2](CLK:= arrSocketMode3StateECS[2] = 'D2', Q=> );
				FPMode3C2[3](CLK:= arrSocketMode3StateECS[3] = 'C2', Q=> );
					FPMode3D2[3](CLK:= arrSocketMode3StateECS[3] = 'D2', Q=> );
						FPMode3C2[4](CLK:= arrSocketMode3StateECS[4] = 'C2', Q=> );
							FPMode3D2[4](CLK:= arrSocketMode3StateECS[4] = 'D2', Q=> );
			
